LIN {X -214.690,Y 120.896,Z -29.506,A 0.015,B -0.000,C -180.000} C_DIS
LIN {X -218.092,Y 115.236,Z -29.750,A 0.015,B 0.000,C -180.000} C_DIS
LIN {X -214.270,Y 109.850,Z -29.994,A 0.015,B 0.000,C 180.000} C_DIS
LIN {X -207.804,Y 111.194,Z -30.238,A 0.015,B 0.000,C 180.000} C_DIS
LIN {X -206.444,Y 117.657,Z -30.482,A 0.015,B 0.000,C 180.000} C_DIS
LIN {X -211.820,Y 121.492,Z -30.726,A 0.015,B 0.000,C 180.000} C_DIS
LIN {X -217.489,Y 118.103,Z -30.970,A 0.015,B 0.000,C -180.000} C_DIS
LIN {X -216.656,Y 111.552,Z -31.214,A 0.015,B -0.000,C -180.000} C_DIS
LIN {X -210.319,Y 109.690,Z -31.458,A 0.015,B 0.000,C -180.000} C_DIS
LIN {X -206.074,Y 114.749,Z -31.702,A 0.015,B 0.000,C 180.000} C_DIS
LIN {X -209.009,Y 120.666,Z -31.946,A 0.015,B 0.000,C 180.000} C_DIS
LIN {X -215.605,Y 120.349,Z -32.190,A 0.015,B -0.000,C 180.000} C_DIS
LIN {X -217.958,Y 114.177,Z -32.435,A 0.015,B 0.000,C -180.000} C_DIS
LIN {X -213.247,Y 109.549,Z -32.679,A 0.015,B 0.000,C 180.000} C_DIS
LIN {X -207.118,Y 112.011,Z -32.923,A 0.015,B 0.000,C 180.000} C_DIS
LIN {X -206.918,Y 118.612,Z -33.167,A 0.015,B 0.000,C -180.000} C_DIS
LIN {X -212.886,Y 121.441,Z -33.411,A 0.015,B 0.000,C -180.000} C_DIS
LIN {X -217.869,Y 117.107,Z -33.655,A 0.015,B -0.000,C 180.000} C_DIS
LIN {X -215.895,Y 110.804,Z -33.899,A 0.015,B 0.000,C 180.000} C_DIS
LIN {X -209.329,Y 110.088,Z -34.143,A 0.015,B 0.000,C -180.000} C_DIS
LIN {X -206.042,Y 115.816,Z -34.387,A 0.015,B 0.000,C -180.000} C_DIS
LIN {X -209.972,Y 121.123,Z -34.631,A 0.015,B 0.000,C -180.000} C_DIS
LIN {X -216.410,Y 119.648,Z -34.875,A 0.015,B -0.000,C -180.000} C_DIS
LIN {X -217.639,Y 113.160,Z -35.119,A 0.015,B 0.000,C -180.000} C_DIS
LIN {X -212.186,Y 109.433,Z -35.363,A 0.015,B 0.000,C 180.000} C_DIS
LIN {X -206.587,Y 112.936,Z -35.607,A 0.015,B 0.000,C 180.000} C_DIS
LIN {X -207.553,Y 119.469,Z -35.851,A 0.015,B 0.000,C -180.000} C_DIS
LIN {X -213.926,Y 121.203,Z -36.095,A 0.015,B 0.000,C 180.000} C_DIS
LIN {X -218.067,Y 116.059,Z -36.339,A 0.015,B 0.000,C -180.000} C_DIS
LIN {X -215.014,Y 110.203,Z -36.583,A 0.015,B -0.000,C -180.000} C_DIS
LIN {X -208.425,Y 110.653,Z -36.827,A 0.015,B 0.000,C 180.000} C_DIS
LIN {X -206.198,Y 116.871,Z -37.071,A 0.015,B 0.000,C 180.000} C_DIS
LIN {X -211.002,Y 121.403,Z -37.315,A 0.015,B 0.000,C -180.000} C_DIS
LIN {X -217.079,Y 118.818,Z -37.560,A 0.015,B 0.000,C 180.000} C_DIS
LIN {X -217.146,Y 112.214,Z -37.804,A 0.015,B -0.000,C 180.000} C_DIS
LIN {X -211.122,Y 109.506,Z -38.048,A 0.015,B -0.000,C 180.000} C_DIS
LIN {X -206.227,Y 113.940,Z -38.292,A 0.015,B -0.000,C 180.000} C_DIS
LIN {X -208.329,Y 120.201,Z -38.536,A 0.015,B 0.000,C 180.000} C_DIS
LIN {X -214.907,Y 120.785,Z -38.780,A 0.015,B 0.000,C -180.000} C_DIS
LIN {X -218.078,Y 114.992,Z -39.024,A 0.015,B 0.000,C 180.000} C_DIS
LIN {X -214.041,Y 109.765,Z -39.268,A 0.015,B 0.000,C -180.000} C_DIS
LIN {X -207.635,Y 111.369,Z -39.512,A 0.015,B -0.000,C 180.000} C_DIS
LIN {X -206.537,Y 117.882,Z -39.756,A 0.015,B 0.000,C -180.000} C_DIS
LIN {X -212.064,Y 121.497,Z -40.000,A 0.015,B -0.000,C 180.000} C_DIS
LIN {X -214.189,Y 121.497,Z -40.000,A 0.015,B 0.000,C 180.000} C_DIS
CIRC {X -216.111,Y 120.388,Z -40.000,A 0.015,B 0.000,C 180.000},{X -216.113,Y 118.169,Z -40.000,A 0.015,B 0.000,C -180.000} C_DIS
LIN {X -214.876,Y 116.023,Z -40.000,A 0.015,B -0.000,C 180.000} C_DIS
CIRC {X -213.837,Y 114.982,Z -40.000,A 0.015,B 0.000,C -180.000},{X -212.416,Y 114.601,Z -40.000,A 0.015,B -0.000,C 180.000} C_DIS
LIN {X -181.082,Y 114.601,Z -40.000,A 0.015,B 0.000,C -180.000} C_DIS
CIRC {X -179.663,Y 114.981,Z -40.000,A 0.015,B -0.000,C -180.000},{X -178.624,Y 116.020,Z -40.000,A 0.015,B 0.000,C -180.000} C_DIS
LIN {X -177.385,Y 118.164,Z -40.000,A 0.015,B -0.000,C 180.000} C_DIS
CIRC {X -177.385,Y 120.386,Z -40.000,A 0.015,B 0.000,C -180.000},{X -179.309,Y 121.497,Z -40.000,A 0.015,B 0.000,C 180.000} C_DIS
LIN {X -212.064,Y 121.497,Z -40.000,A 0.015,B -0.000,C 180.000} C_DIS
CIRC {X -215.504,Y 122.547,Z -40.000,A 0.015,B 0.000,C -180.000},{X -217.770,Y 125.339,Z -40.000,A 0.015,B 0.000,C 180.000} C_DIS
CIRC {X -219.938,Y 128.171,Z -40.000,A 0.015,B -0.000,C 180.000},{X -223.248,Y 129.500,Z -40.000,A 0.015,B -0.000,C -180.000} C_DIS
CIRC {X -226.517,Y 129.867,Z -40.000,A 0.015,B 0.000,C -180.000},{X -229.788,Y 130.221,Z -40.000,A 0.015,B 0.000,C 180.000} C_DIS
CIRC {X -231.585,Y 129.305,Z -40.000,A 0.015,B -0.000,C 180.000},{X -231.476,Y 127.292,Z -40.000,A 0.015,B -0.000,C -180.000} C_DIS
CIRC {X -228.692,Y 123.319,Z -40.000,A 0.015,B 0.000,C -180.000},{X -226.063,Y 119.242,Z -40.000,A 0.015,B 0.000,C 180.000} C_DIS
CIRC {X -223.545,Y 115.096,Z -40.000,A 0.015,B 0.000,C 180.000},{X -221.091,Y 110.912,Z -40.000,A 0.015,B 0.000,C -180.000} C_DIS
CIRC {X -217.986,Y 107.803,Z -40.000,A 0.015,B 0.000,C 180.000},{X -213.742,Y 106.665,Z -40.000,A 0.015,B 0.000,C 180.000} C_DIS
LIN {X -179.770,Y 106.665,Z -40.000,A 0.015,B 0.000,C -180.000} C_DIS
CIRC {X -175.521,Y 107.803,Z -40.000,A 0.015,B 0.000,C 180.000},{X -172.409,Y 110.912,Z -40.000,A 0.015,B 0.000,C 180.000} C_DIS
CIRC {X -169.958,Y 115.089,Z -40.000,A 0.015,B -0.000,C -180.000},{X -167.450,Y 119.233,Z -40.000,A 0.015,B 0.000,C 180.000} C_DIS
CIRC {X -164.835,Y 123.311,Z -40.000,A 0.015,B 0.000,C -180.000},{X -162.065,Y 127.285,Z -40.000,A 0.015,B 0.000,C -180.000} C_DIS
CIRC {X -161.960,Y 129.301,Z -40.000,A 0.015,B 0.000,C 180.000},{X -163.759,Y 130.217,Z -40.000,A 0.015,B -0.000,C 180.000} C_DIS
CIRC {X -167.466,Y 129.816,Z -40.000,A 0.015,B 0.000,C -180.000},{X -171.172,Y 129.397,Z -40.000,A 0.015,B 0.000,C -180.000} C_DIS
CIRC {X -174.888,Y 129.076,Z -40.000,A 0.015,B 0.000,C 180.000},{X -178.617,Y 128.969,Z -40.000,A 0.015,B 0.000,C -180.000} C_DIS
LIN {X -214.895,Y 128.968,Z -40.000,A 0.015,B 0.000,C -180.000} C_DIS
CIRC {X -218.633,Y 129.075,Z -40.000,A 0.015,B 0.000,C -180.000},{X -222.358,Y 129.398,Z -40.000,A 0.015,B -0.000,C -180.000} C_DIS
LIN {X -223.248,Y 129.500,Z -40.000,A 0.015,B 0.000,C 180.000} C_DIS
CIRC {X -226.419,Y 130.853,Z -40.000,A 0.015,B 0.000,C 180.000},{X -228.335,Y 133.719,Z -40.000,A 0.015,B -0.000,C 180.000} C_DIS
CIRC {X -230.253,Y 136.582,Z -40.000,A 0.015,B 0.000,C -180.000},{X -233.421,Y 137.938,Z -40.000,A 0.015,B 0.000,C -180.000} C_DIS
CIRC {X -237.034,Y 138.381,Z -40.000,A 0.015,B 0.000,C 180.000},{X -240.642,Y 138.863,Z -40.000,A 0.015,B 0.000,C 180.000} C_DIS
CIRC {X -242.321,Y 139.135,Z -40.000,A 0.015,B 0.000,C -180.000},{X -243.987,Y 139.480,Z -40.000,A 0.015,B 0.000,C 180.000} C_DIS
CIRC {X -245.648,Y 139.845,Z -40.000,A 0.015,B -0.000,C -180.000},{X -247.316,Y 140.180,Z -40.000,A 0.015,B 0.000,C 180.000} C_DIS
CIRC {X -249.035,Y 139.393,Z -40.000,A 0.015,B 0.000,C -180.000},{X -248.855,Y 137.511,Z -40.000,A 0.015,B -0.000,C -180.000} C_DIS
LIN {X -243.268,Y 131.116,Z -40.000,A 0.015,B 0.000,C -180.000} C_DIS
CIRC {X -240.525,Y 127.874,Z -40.000,A 0.015,B -0.000,C 180.000},{X -237.914,Y 124.524,Z -40.000,A 0.015,B 0.000,C -180.000} C_DIS
CIRC {X -234.428,Y 119.496,Z -40.000,A 0.015,B -0.000,C -180.000},{X -231.314,Y 114.230,Z -40.000,A 0.015,B -0.000,C -180.000} C_DIS
CIRC {X -228.360,Y 108.876,Z -40.000,A 0.015,B 0.000,C -180.000},{X -225.339,Y 103.559,Z -40.000,A 0.015,B -0.000,C -180.000} C_DIS
CIRC {X -222.234,Y 100.451,Z -40.000,A 0.015,B -0.000,C -180.000},{X -217.991,Y 99.313,Z -40.000,A 0.015,B 0.000,C -180.000} C_DIS
LIN {X -175.527,Y 99.313,Z -40.000,A 0.015,B 0.000,C 180.000} C_DIS
CIRC {X -171.278,Y 100.451,Z -40.000,A 0.015,B 0.000,C 180.000},{X -168.166,Y 103.560,Z -40.000,A 0.015,B 0.000,C -180.000} C_DIS
CIRC {X -167.080,Y 105.510,Z -40.000,A 0.015,B 0.000,C -180.000},{X -166.055,Y 107.493,Z -40.000,A 0.015,B 0.000,C 180.000} C_DIS
CIRC {X -165.030,Y 109.476,Z -40.000,A 0.015,B -0.000,C 180.000},{X -163.943,Y 111.426,Z -40.000,A 0.015,B 0.000,C 180.000} C_DIS
CIRC {X -159.653,Y 118.326,Z -40.000,A 0.015,B 0.000,C 180.000},{X -154.928,Y 124.936,Z -40.000,A 0.015,B -0.000,C 180.000} C_DIS
CIRC {X -149.891,Y 131.308,Z -40.000,A 0.015,B -0.000,C 180.000},{X -144.653,Y 137.515,Z -40.000,A 0.015,B 0.000,C 180.000} C_DIS
CIRC {X -144.469,Y 139.395,Z -40.000,A 0.015,B 0.000,C -180.000},{X -146.185,Y 140.182,Z -40.000,A 0.015,B 0.000,C 180.000} C_DIS
CIRC {X -169.667,Y 136.815,Z -40.000,A 0.015,B 0.000,C -180.000},{X -193.359,Y 135.650,Z -40.000,A 0.015,B -0.000,C 180.000} C_DIS
CIRC {X -213.424,Y 136.197,Z -40.000,A 0.015,B -0.000,C 180.000},{X -233.421,Y 137.938,Z -40.000,A 0.015,B 0.000,C -180.000} C_DIS
CIRC {X -236.184,Y 139.158,Z -40.000,A 0.015,B 0.000,C 180.000},{X -237.779,Y 141.722,Z -40.000,A 0.015,B -0.000,C -180.000} C_DIS
CIRC {X -239.318,Y 144.301,Z -40.000,A 0.015,B 0.000,C -180.000},{X -241.992,Y 145.667,Z -40.000,A 0.015,B 0.000,C -180.000} C_DIS
CIRC {X -243.728,Y 146.016,Z -40.000,A 0.015,B 0.000,C 180.000},{X -245.460,Y 146.386,Z -40.000,A 0.015,B 0.000,C 180.000} C_DIS
CIRC {X -260.324,Y 150.371,Z -40.000,A 0.015,B -0.000,C 180.000},{X -274.770,Y 155.672,Z -40.000,A 0.015,B 0.000,C 180.000} C_DIS
CIRC {X -276.326,Y 155.146,Z -40.000,A 0.015,B 0.000,C -180.000},{X -275.997,Y 153.536,Z -40.000,A 0.015,B 0.000,C -180.000} C_DIS
CIRC {X -266.962,Y 146.173,Z -40.000,A 0.015,B 0.000,C -180.000},{X -258.508,Y 138.148,Z -40.000,A 0.015,B 0.000,C -180.000} C_DIS
CIRC {X -250.643,Y 129.549,Z -40.000,A 0.015,B 0.000,C 180.000},{X -243.360,Y 120.451,Z -40.000,A 0.015,B 0.000,C 180.000} C_DIS
CIRC {X -241.141,Y 117.355,Z -40.000,A 0.015,B 0.000,C -180.000},{X -239.047,Y 114.173,Z -40.000,A 0.015,B 0.000,C -180.000} C_DIS
CIRC {X -237.049,Y 110.931,Z -40.000,A 0.015,B 0.000,C -180.000},{X -235.115,Y 107.650,Z -40.000,A 0.015,B -0.000,C 180.000} C_DIS
CIRC {X -233.613,Y 104.946,Z -40.000,A 0.015,B -0.000,C 180.000},{X -232.196,Y 102.197,Z -40.000,A 0.015,B -0.000,C -180.000} C_DIS
CIRC {X -230.779,Y 99.448,Z -40.000,A 0.015,B 0.000,C -180.000},{X -229.277,Y 96.745,Z -40.000,A 0.015,B -0.000,C -180.000} C_DIS
CIRC {X -226.172,Y 93.636,Z -40.000,A 0.015,B -0.000,C -180.000},{X -221.929,Y 92.498,Z -40.000,A 0.015,B 0.000,C 180.000} C_DIS
LIN {X -171.595,Y 92.498,Z -40.000,A 0.015,B -0.000,C 180.000} C_DIS
CIRC {X -167.346,Y 93.636,Z -40.000,A 0.015,B 0.000,C 180.000},{X -164.234,Y 96.746,Z -40.000,A 0.015,B 0.000,C -180.000} C_DIS
CIRC {X -162.669,Y 99.555,Z -40.000,A 0.015,B -0.000,C 180.000},{X -161.192,Y 102.412,Z -40.000,A 0.015,B -0.000,C -180.000} C_DIS
CIRC {X -159.715,Y 105.268,Z -40.000,A 0.015,B 0.000,C 180.000},{X -158.150,Y 108.078,Z -40.000,A 0.015,B 0.000,C 180.000} C_DIS
CIRC {X -149.768,Y 120.946,Z -40.000,A 0.015,B 0.000,C -180.000},{X -140.064,Y 132.849,Z -40.000,A 0.015,B -0.000,C 180.000} C_DIS
CIRC {X -129.235,Y 143.731,Z -40.000,A 0.015,B 0.000,C 180.000},{X -117.456,Y 153.577,Z -40.000,A 0.015,B 0.000,C 180.000} C_DIS
CIRC {X -117.135,Y 155.187,Z -40.000,A 0.015,B 0.000,C -180.000},{X -118.693,Y 155.704,Z -40.000,A 0.015,B 0.000,C -180.000} C_DIS
CIRC {X -128.956,Y 151.768,Z -40.000,A 0.015,B -0.000,C 180.000},{X -139.478,Y 148.589,Z -40.000,A 0.015,B 0.000,C 180.000} C_DIS
CIRC {X -150.185,Y 146.112,Z -40.000,A 0.015,B 0.000,C 180.000},{X -161.020,Y 144.276,Z -40.000,A 0.015,B 0.000,C 180.000} C_DIS
CIRC {X -169.797,Y 143.362,Z -40.000,A 0.015,B -0.000,C -180.000},{X -178.617,Y 143.057,Z -40.000,A 0.015,B -0.000,C -180.000} C_DIS
LIN {X -214.895,Y 143.057,Z -40.000,A 0.015,B 0.000,C 180.000} C_DIS
CIRC {X -228.506,Y 143.711,Z -40.000,A 0.015,B 0.000,C 180.000},{X -241.992,Y 145.667,Z -40.000,A 0.015,B 0.000,C -180.000} C_DIS
CIRC {X -244.741,Y 147.123,Z -40.000,A 0.015,B 0.000,C 180.000},{X -246.215,Y 149.862,Z -40.000,A 0.015,B 0.000,C -180.000} C_DIS
CIRC {X -247.650,Y 152.609,Z -40.000,A 0.015,B 0.000,C 180.000},{X -250.334,Y 154.160,Z -40.000,A 0.015,B 0.000,C 180.000} C_DIS
CIRC {X -257.545,Y 156.101,Z -40.000,A 0.015,B -0.000,C 180.000},{X -264.665,Y 158.353,Z -40.000,A 0.015,B 0.000,C -180.000} C_DIS
CIRC {X -269.256,Y 160.100,Z -40.000,A 0.015,B 0.000,C 180.000},{X -273.710,Y 162.168,Z -40.000,A 0.015,B -0.000,C -180.000} C_DIS
LIN {X -283.276,Y 167.029,Z -40.000,A 0.015,B -0.000,C -180.000} C_DIS
CIRC {X -285.545,Y 166.939,Z -40.000,A 0.015,B 0.000,C 180.000},{X -286.654,Y 164.957,Z -40.000,A 0.015,B 0.000,C -180.000} C_DIS
LIN {X -286.654,Y 156.539,Z -40.000,A 0.015,B 0.000,C -180.000} C_DIS
CIRC {X -285.883,Y 153.392,Z -40.000,A 0.015,B 0.000,C 180.000},{X -283.747,Y 150.958,Z -40.000,A 0.015,B 0.000,C 180.000} C_DIS
CIRC {X -271.170,Y 141.133,Z -40.000,A 0.015,B 0.000,C -180.000},{X -259.697,Y 130.038,Z -40.000,A 0.015,B 0.000,C -180.000} C_DIS
CIRC {X -249.502,Y 117.754,Z -40.000,A 0.015,B 0.000,C -180.000},{X -240.761,Y 104.396,Z -40.000,A 0.015,B 0.000,C 180.000} C_DIS
CIRC {X -238.793,Y 100.854,Z -40.000,A 0.015,B 0.000,C 180.000},{X -236.936,Y 97.253,Z -40.000,A 0.015,B 0.000,C 180.000} C_DIS
CIRC {X -235.080,Y 93.651,Z -40.000,A 0.015,B -0.000,C -180.000},{X -233.112,Y 90.109,Z -40.000,A 0.015,B 0.000,C -180.000} C_DIS
CIRC {X -230.007,Y 87.001,Z -40.000,A 0.015,B 0.000,C 180.000},{X -225.763,Y 85.863,Z -40.000,A 0.015,B 0.000,C 180.000} C_DIS
LIN {X -167.766,Y 85.863,Z -40.000,A 0.015,B 0.000,C 180.000} C_DIS
CIRC {X -163.516,Y 87.001,Z -40.000,A 0.015,B 0.000,C 180.000},{X -160.405,Y 90.110,Z -40.000,A 0.015,B 0.000,C 180.000} C_DIS
CIRC {X -158.373,Y 93.756,Z -40.000,A 0.015,B 0.000,C 180.000},{X -156.456,Y 97.464,Z -40.000,A 0.015,B 0.000,C -180.000} C_DIS
CIRC {X -154.540,Y 101.171,Z -40.000,A 0.015,B 0.000,C -180.000},{X -152.508,Y 104.817,Z -40.000,A 0.015,B 0.000,C 180.000} C_DIS
CIRC {X -143.805,Y 118.066,Z -40.000,A 0.015,B 0.000,C -180.000},{X -133.646,Y 130.234,Z -40.000,A 0.015,B -0.000,C 180.000} C_DIS
CIRC {X -122.233,Y 141.226,Z -40.000,A 0.015,B 0.000,C -180.000},{X -109.753,Y 150.992,Z -40.000,A 0.015,B 0.000,C 180.000} C_DIS
CIRC {X -107.625,Y 153.424,Z -40.000,A 0.015,B 0.000,C 180.000},{X -106.858,Y 156.564,Z -40.000,A 0.015,B -0.000,C 180.000} C_DIS
LIN {X -106.859,Y 164.937,Z -40.000,A 0.015,B 0.000,C -180.000} C_DIS
CIRC {X -107.968,Y 166.911,Z -40.000,A 0.015,B 0.000,C 180.000},{X -110.230,Y 166.990,Z -40.000,A 0.015,B -0.000,C 180.000} C_DIS
CIRC {X -122.583,Y 161.292,Z -40.000,A 0.015,B 0.000,C 180.000},{X -135.397,Y 156.724,Z -40.000,A 0.015,B -0.000,C -180.000} C_DIS
CIRC {X -148.548,Y 153.257,Z -40.000,A 0.015,B 0.000,C -180.000},{X -161.934,Y 150.848,Z -40.000,A 0.015,B 0.000,C 180.000} C_DIS
CIRC {X -170.255,Y 149.982,Z -40.000,A 0.015,B 0.000,C 180.000},{X -178.617,Y 149.693,Z -40.000,A 0.015,B 0.000,C -180.000} C_DIS
LIN {X -214.895,Y 149.693,Z -40.000,A 0.015,B 0.000,C 180.000} C_DIS
CIRC {X -227.567,Y 150.265,Z -40.000,A 0.015,B -0.000,C -180.000},{X -240.136,Y 151.977,Z -40.000,A 0.015,B 0.000,C -180.000} C_DIS
CIRC {X -245.252,Y 152.991,Z -40.000,A 0.015,B 0.000,C 180.000},{X -250.334,Y 154.160,Z -40.000,A 0.015,B -0.000,C 180.000} C_DIS
CIRC {X -253.660,Y 156.157,Z -40.000,A 0.015,B -0.000,C 180.000},{X -255.280,Y 159.681,Z -40.000,A 0.015,B -0.000,C -180.000} C_DIS
CIRC {X -256.805,Y 163.218,Z -40.000,A 0.015,B 0.000,C 180.000},{X -259.959,Y 165.430,Z -40.000,A 0.015,B -0.000,C 180.000} C_DIS
CIRC {X -276.245,Y 172.320,Z -40.000,A 0.015,B 0.000,C 180.000},{X -291.506,Y 181.253,Z -40.000,A 0.015,B 0.000,C -180.000} C_DIS
CIRC {X -293.652,Y 181.365,Z -40.000,A 0.015,B -0.000,C -180.000},{X -294.758,Y 179.523,Z -40.000,A 0.015,B 0.000,C 180.000} C_DIS
LIN {X -294.757,Y 153.804,Z -40.000,A 0.015,B 0.000,C 180.000} C_DIS
CIRC {X -293.661,Y 149.334,Z -40.000,A 0.015,B -0.000,C -180.000},{X -290.622,Y 145.877,Z -40.000,A 0.015,B 0.000,C 180.000} C_DIS
CIRC {X -286.379,Y 142.894,Z -40.000,A 0.015,B 0.000,C 180.000},{X -282.158,Y 139.879,Z -40.000,A 0.015,B 0.000,C 180.000} C_DIS
CIRC {X -278.036,Y 136.728,Z -40.000,A 0.015,B 0.000,C -180.000},{X -274.099,Y 133.347,Z -40.000,A 0.015,B -0.000,C 180.000} C_DIS
CIRC {X -268.929,Y 128.312,Z -40.000,A 0.015,B -0.000,C -180.000},{X -264.114,Y 122.936,Z -40.000,A 0.015,B 0.000,C 180.000} C_DIS
CIRC {X -259.562,Y 117.340,Z -40.000,A 0.015,B 0.000,C 180.000},{X -255.164,Y 111.623,Z -40.000,A 0.015,B 0.000,C -180.000} C_DIS
CIRC {X -251.289,Y 106.107,Z -40.000,A 0.015,B 0.000,C 180.000},{X -247.750,Y 100.369,Z -40.000,A 0.015,B 0.000,C -180.000} C_DIS
CIRC {X -245.202,Y 95.810,Z -40.000,A 0.015,B -0.000,C 180.000},{X -242.773,Y 91.187,Z -40.000,A 0.015,B 0.000,C 180.000} C_DIS
CIRC {X -240.344,Y 86.564,Z -40.000,A 0.015,B 0.000,C -180.000},{X -237.795,Y 82.006,Z -40.000,A 0.015,B -0.000,C -180.000} C_DIS
CIRC {X -234.690,Y 78.897,Z -40.000,A 0.015,B 0.000,C -180.000},{X -230.446,Y 77.759,Z -40.000,A 0.015,B 0.000,C 180.000} C_DIS
LIN {X -163.089,Y 77.759,Z -40.000,A 0.015,B 0.000,C 180.000} C_DIS
CIRC {X -158.840,Y 78.897,Z -40.000,A 0.015,B 0.000,C -180.000},{X -155.728,Y 82.007,Z -40.000,A 0.015,B 0.000,C -180.000} C_DIS
CIRC {X -153.114,Y 86.666,Z -40.000,A 0.015,B 0.000,C -180.000},{X -150.619,Y 91.390,Z -40.000,A 0.015,B -0.000,C 180.000} C_DIS
CIRC {X -148.124,Y 96.114,Z -40.000,A 0.015,B -0.000,C 180.000},{X -145.510,Y 100.773,Z -40.000,A 0.015,B 0.000,C 180.000} C_DIS
CIRC {X -136.917,Y 113.796,Z -40.000,A 0.015,B 0.000,C -180.000},{X -126.846,Y 125.713,Z -40.000,A 0.015,B 0.000,C 180.000} C_DIS
CIRC {X -115.486,Y 136.403,Z -40.000,A 0.015,B 0.000,C -180.000},{X -103.022,Y 145.783,Z -40.000,A 0.015,B 0.000,C 180.000} C_DIS
CIRC {X -99.888,Y 149.247,Z -40.000,A 0.015,B 0.000,C -180.000},{X -98.755,Y 153.779,Z -40.000,A 0.015,B 0.000,C -180.000} C_DIS
LIN {X -98.755,Y 179.510,Z -40.000,A 0.015,B 0.000,C 180.000} C_DIS
CIRC {X -99.862,Y 181.369,Z -40.000,A 0.015,B 0.000,C 180.000},{X -102.023,Y 181.282,Z -40.000,A 0.015,B 0.000,C -180.000} C_DIS
CIRC {X -110.211,Y 176.258,Z -40.000,A 0.015,B 0.000,C 180.000},{X -118.658,Y 171.685,Z -40.000,A 0.015,B -0.000,C 180.000} C_DIS
CIRC {X -127.391,Y 167.675,Z -40.000,A 0.015,B 0.000,C 180.000},{X -136.407,Y 164.351,Z -40.000,A 0.015,B 0.000,C -180.000} C_DIS
CIRC {X -155.656,Y 159.675,Z -40.000,A 0.015,B 0.000,C -180.000},{X -175.393,Y 157.980,Z -40.000,A 0.015,B 0.000,C -180.000} C_DIS
LIN {X -214.895,Y 157.797,Z -40.000,A 0.015,B -0.000,C 180.000} C_DIS
CIRC {X -237.748,Y 159.718,Z -40.000,A 0.015,B -0.000,C 180.000},{X -259.959,Y 165.430,Z -40.000,A 0.015,B 0.000,C 180.000} C_DIS
CIRC {X -262.962,Y 167.626,Z -40.000,A 0.015,B -0.000,C 180.000},{X -264.228,Y 171.125,Z -40.000,A 0.015,B 0.000,C -180.000} C_DIS
CIRC {X -265.425,Y 174.627,Z -40.000,A 0.015,B 0.000,C 180.000},{X -268.291,Y 176.970,Z -40.000,A 0.015,B 0.000,C 180.000} C_DIS
CIRC {X -272.041,Y 178.652,Z -40.000,A 0.015,B 0.000,C 180.000},{X -275.743,Y 180.440,Z -40.000,A 0.015,B 0.000,C 180.000} C_DIS
CIRC {X -282.030,Y 183.929,Z -40.000,A 0.015,B 0.000,C 180.000},{X -287.996,Y 187.941,Z -40.000,A 0.015,B 0.000,C -180.000} C_DIS
CIRC {X -293.740,Y 192.257,Z -40.000,A 0.015,B 0.000,C 180.000},{X -299.397,Y 196.684,Z -40.000,A 0.015,B 0.000,C 180.000} C_DIS
CIRC {X -301.459,Y 196.918,Z -40.000,A 0.015,B 0.000,C 180.000},{X -302.564,Y 195.161,Z -40.000,A 0.015,B -0.000,C -180.000} C_DIS
LIN {X -302.562,Y 149.253,Z -40.000,A 0.015,B 0.000,C -180.000} C_DIS
CIRC {X -301.466,Y 144.963,Z -40.000,A 0.015,B 0.000,C -180.000},{X -298.447,Y 141.724,Z -40.000,A 0.015,B 0.000,C 180.000} C_DIS
CIRC {X -288.038,Y 134.334,Z -40.000,A 0.015,B -0.000,C 180.000},{X -278.369,Y 125.999,Z -40.000,A 0.015,B 0.000,C 180.000} C_DIS
CIRC {X -269.486,Y 116.835,Z -40.000,A 0.015,B -0.000,C 180.000},{X -261.414,Y 106.948,Z -40.000,A 0.015,B 0.000,C 180.000} C_DIS
CIRC {X -257.807,Y 101.813,Z -40.000,A 0.015,B 0.000,C 180.000},{X -254.513,Y 96.472,Z -40.000,A 0.015,B 0.000,C 180.000} C_DIS
CIRC {X -251.402,Y 90.936,Z -40.000,A 0.015,B -0.000,C -180.000},{X -248.409,Y 85.336,Z -40.000,A 0.015,B -0.000,C 180.000} C_DIS
CIRC {X -245.417,Y 79.736,Z -40.000,A 0.015,B -0.000,C 180.000},{X -242.306,Y 74.201,Z -40.000,A 0.015,B 0.000,C 180.000} C_DIS
CIRC {X -239.201,Y 71.092,Z -40.000,A 0.015,B 0.000,C -180.000},{X -234.957,Y 69.954,Z -40.000,A 0.015,B 0.000,C 180.000} C_DIS
LIN {X -158.585,Y 69.954,Z -40.000,A 0.015,B 0.000,C 180.000} C_DIS
CIRC {X -154.336,Y 71.092,Z -40.000,A 0.015,B 0.000,C 180.000},{X -151.224,Y 74.201,Z -40.000,A 0.015,B -0.000,C 180.000} C_DIS
LIN {X -138.752,Y 96.868,Z -40.000,A 0.015,B -0.000,C -180.000} C_DIS
CIRC {X -130.141,Y 109.762,Z -40.000,A 0.015,B 0.000,C -180.000},{X -119.937,Y 121.436,Z -40.000,A 0.015,B 0.000,C 180.000} C_DIS
CIRC {X -108.478,Y 131.862,Z -40.000,A 0.015,B 0.000,C 180.000},{X -96.045,Y 141.103,Z -40.000,A 0.015,B 0.000,C -180.000} C_DIS
LIN {X -95.557,Y 141.407,Z -40.000,A 0.015,B -0.000,C 180.000} C_DIS
LIN {X -95.066,Y 141.708,Z -40.000,A 0.015,B 0.000,C 180.000} C_DIS
CIRC {X -92.045,Y 144.990,Z -40.000,A 0.015,B 0.000,C 180.000},{X -90.949,Y 149.315,Z -40.000,A 0.015,B 0.000,C 180.000} C_DIS
LIN {X -90.951,Y 195.181,Z -40.000,A 0.015,B 0.000,C 180.000} C_DIS
CIRC {X -92.055,Y 196.943,Z -40.000,A 0.015,B -0.000,C 180.000},{X -94.122,Y 196.716,Z -40.000,A 0.015,B 0.000,C 180.000} C_DIS
CIRC {X -101.310,Y 191.252,Z -40.000,A 0.015,B 0.000,C -180.000},{X -108.704,Y 186.071,Z -40.000,A 0.015,B -0.000,C 180.000} C_DIS
CIRC {X -116.396,Y 181.333,Z -40.000,A 0.015,B -0.000,C 180.000},{X -124.441,Y 177.222,Z -40.000,A 0.015,B 0.000,C 180.000} C_DIS
CIRC {X -134.001,Y 173.361,Z -40.000,A 0.015,B -0.000,C 180.000},{X -143.892,Y 170.451,Z -40.000,A 0.015,B 0.000,C 180.000} C_DIS
CIRC {X -153.962,Y 168.277,Z -40.000,A 0.015,B 0.000,C 180.000},{X -164.126,Y 166.605,Z -40.000,A 0.015,B 0.000,C 180.000} C_DIS
CIRC {X -171.354,Y 165.853,Z -40.000,A 0.015,B 0.000,C -180.000},{X -178.617,Y 165.602,Z -40.000,A 0.015,B 0.000,C -180.000} C_DIS
LIN {X -214.895,Y 165.602,Z -40.000,A 0.015,B 0.000,C 180.000} C_DIS
CIRC {X -230.659,Y 166.574,Z -40.000,A 0.015,B 0.000,C 180.000},{X -246.184,Y 169.475,Z -40.000,A 0.015,B -0.000,C -180.000} C_DIS
CIRC {X -257.388,Y 172.777,Z -40.000,A 0.015,B 0.000,C 180.000},{X -268.291,Y 176.970,Z -40.000,A 0.015,B 0.000,C 180.000} C_DIS
CIRC {X -271.061,Y 179.343,Z -40.000,A 0.015,B -0.000,C -180.000},{X -272.000,Y 182.868,Z -40.000,A 0.015,B 0.000,C -180.000} C_DIS
CIRC {X -272.841,Y 186.389,Z -40.000,A 0.015,B 0.000,C 180.000},{X -275.400,Y 188.950,Z -40.000,A 0.015,B 0.000,C -180.000} C_DIS
CIRC {X -292.319,Y 200.359,Z -40.000,A 0.015,B -0.000,C -180.000},{X -307.135,Y 214.394,Z -40.000,A 0.015,B 0.000,C 180.000} C_DIS
CIRC {X -309.015,Y 214.857,Z -40.000,A 0.015,B 0.000,C 180.000},{X -310.116,Y 213.263,Z -40.000,A 0.015,B -0.000,C -180.000} C_DIS
LIN {X -310.114,Y 144.714,Z -40.000,A 0.015,B 0.000,C -180.000} C_DIS
CIRC {X -309.001,Y 140.539,Z -40.000,A 0.015,B -0.000,C 180.000},{X -305.958,Y 137.471,Z -40.000,A 0.015,B -0.000,C -180.000} C_DIS
CIRC {X -295.027,Y 130.251,Z -40.000,A 0.015,B 0.000,C 180.000},{X -284.953,Y 121.878,Z -40.000,A 0.015,B -0.000,C 180.000} C_DIS
CIRC {X -275.768,Y 112.547,Z -40.000,A 0.015,B 0.000,C 180.000},{X -267.461,Y 102.426,Z -40.000,A 0.015,B 0.000,C 180.000} C_DIS
CIRC {X -264.114,Y 97.659,Z -40.000,A 0.015,B 0.000,C -180.000},{X -261.056,Y 92.701,Z -40.000,A 0.015,B -0.000,C 180.000} C_DIS
LIN {X -246.670,Y 66.649,Z -40.000,A 0.015,B 0.000,C -180.000} C_DIS
CIRC {X -243.565,Y 63.540,Z -40.000,A 0.015,B 0.000,C -180.000},{X -239.321,Y 62.402,Z -40.000,A 0.015,B 0.000,C 180.000} C_DIS
LIN {X -154.227,Y 62.402,Z -40.000,A 0.015,B -0.000,C 180.000} C_DIS
CIRC {X -149.978,Y 63.540,Z -40.000,A 0.015,B 0.000,C 180.000},{X -146.866,Y 66.650,Z -40.000,A 0.015,B 0.000,C 180.000} C_DIS
LIN {X -132.214,Y 93.089,Z -40.000,A 0.015,B 0.000,C -180.000} C_DIS
CIRC {X -123.318,Y 106.303,Z -40.000,A 0.015,B 0.000,C 180.000},{X -112.701,Y 118.178,Z -40.000,A 0.015,B 0.000,C 180.000} C_DIS
CIRC {X -100.668,Y 128.600,Z -40.000,A 0.015,B 0.000,C -180.000},{X -87.492,Y 137.534,Z -40.000,A 0.015,B -0.000,C -180.000} C_DIS
CIRC {X -84.493,Y 140.594,Z -40.000,A 0.015,B 0.000,C -180.000},{X -83.398,Y 144.736,Z -40.000,A 0.015,B 0.000,C -180.000} C_DIS
LIN {X -83.400,Y 213.259,Z -40.000,A 0.015,B 0.000,C -180.000} C_DIS
CIRC {X -84.500,Y 214.853,Z -40.000,A 0.015,B 0.000,C 180.000},{X -86.381,Y 214.390,Z -40.000,A 0.015,B -0.000,C 180.000} C_DIS
CIRC {X -98.149,Y 202.832,Z -40.000,A 0.015,B 0.000,C 180.000},{X -111.404,Y 193.014,Z -40.000,A 0.015,B 0.000,C -180.000} C_DIS
CIRC {X -125.835,Y 185.039,Z -40.000,A 0.015,B 0.000,C -180.000},{X -141.159,Y 178.954,Z -40.000,A 0.015,B 0.000,C -180.000} C_DIS
CIRC {X -159.214,Y 174.612,Z -40.000,A 0.015,B 0.000,C 180.000},{X -177.725,Y 173.153,Z -40.000,A 0.015,B 0.000,C 180.000} C_DIS
LIN {X -214.895,Y 173.153,Z -40.000,A 0.015,B 0.000,C 180.000} C_DIS
CIRC {X -246.162,Y 177.168,Z -40.000,A 0.015,B 0.000,C 180.000},{X -275.400,Y 188.950,Z -40.000,A 0.015,B -0.000,C 180.000} C_DIS
CIRC {X -277.772,Y 191.437,Z -40.000,A 0.015,B 0.000,C -180.000},{X -278.335,Y 194.828,Z -40.000,A 0.015,B 0.000,C 180.000} C_DIS
CIRC {X -278.819,Y 198.208,Z -40.000,A 0.015,B 0.000,C 180.000},{X -281.003,Y 200.832,Z -40.000,A 0.015,B 0.000,C 180.000} C_DIS
CIRC {X -299.481,Y 216.465,Z -40.000,A 0.015,B 0.000,C 180.000},{X -314.434,Y 235.497,Z -40.000,A 0.015,B 0.000,C 180.000} C_DIS
CIRC {X -316.141,Y 236.143,Z -40.000,A 0.015,B 0.000,C -180.000},{X -317.237,Y 234.683,Z -40.000,A 0.015,B 0.000,C -180.000} C_DIS
LIN {X -317.235,Y 140.248,Z -40.000,A 0.015,B 0.000,C -180.000} C_DIS
CIRC {X -316.140,Y 136.253,Z -40.000,A 0.015,B 0.000,C 180.000},{X -313.163,Y 133.373,Z -40.000,A 0.015,B -0.000,C -180.000} C_DIS
CIRC {X -302.924,Y 127.100,Z -40.000,A 0.015,B 0.000,C 180.000},{X -293.337,Y 119.870,Z -40.000,A 0.015,B 0.000,C 180.000} C_DIS
CIRC {X -284.520,Y 111.716,Z -40.000,A 0.015,B 0.000,C -180.000},{X -276.595,Y 102.693,Z -40.000,A 0.015,B 0.000,C 180.000} C_DIS
CIRC {X -269.249,Y 92.450,Z -40.000,A 0.015,B 0.000,C 180.000},{X -262.891,Y 81.566,Z -40.000,A 0.015,B 0.000,C -180.000} C_DIS
CIRC {X -256.941,Y 70.468,Z -40.000,A 0.015,B 0.000,C -180.000},{X -250.766,Y 59.494,Z -40.000,A 0.015,B 0.000,C -180.000} C_DIS
CIRC {X -247.686,Y 56.410,Z -40.000,A 0.015,B 0.000,C -180.000},{X -243.475,Y 55.281,Z -40.000,A 0.015,B 0.000,C -180.000} C_DIS
LIN {X -150.053,Y 55.281,Z -40.000,A 0.015,B 0.000,C 180.000} C_DIS
CIRC {X -145.860,Y 56.404,Z -40.000,A 0.015,B 0.000,C -180.000},{X -142.789,Y 59.473,Z -40.000,A 0.015,B -0.000,C 180.000} C_DIS
LIN {X -126.048,Y 89.526,Z -40.000,A 0.015,B 0.000,C -180.000} C_DIS
CIRC {X -117.054,Y 102.798,Z -40.000,A 0.015,B 0.000,C 180.000},{X -106.258,Y 114.650,Z -40.000,A 0.015,B -0.000,C -180.000} C_DIS
CIRC {X -93.931,Y 124.893,Z -40.000,A 0.015,B 0.000,C 180.000},{X -80.345,Y 133.396,Z -40.000,A 0.015,B 0.000,C -180.000} C_DIS
CIRC {X -77.371,Y 136.233,Z -40.000,A 0.015,B -0.000,C 180.000},{X -76.276,Y 140.194,Z -40.000,A 0.015,B 0.000,C -180.000} C_DIS
LIN {X -76.279,Y 234.676,Z -40.000,A 0.015,B 0.000,C 180.000} C_DIS
CIRC {X -77.375,Y 236.136,Z -40.000,A 0.015,B 0.000,C -180.000},{X -79.083,Y 235.489,Z -40.000,A 0.015,B 0.000,C -180.000} C_DIS
CIRC {X -106.859,Y 204.970,Z -40.000,A 0.015,B 0.000,C 180.000},{X -143.363,Y 185.725,Z -40.000,A 0.015,B 0.000,C -180.000} C_DIS
CIRC {X -160.917,Y 181.529,Z -40.000,A 0.015,B 0.000,C -180.000},{X -178.914,Y 180.181,Z -40.000,A 0.015,B 0.000,C 180.000} C_DIS
LIN {X -214.895,Y 180.275,Z -40.000,A 0.015,B 0.000,C 180.000} C_DIS
CIRC {X -244.278,Y 184.041,Z -40.000,A 0.015,B 0.000,C -180.000},{X -271.760,Y 195.096,Z -40.000,A 0.015,B 0.000,C -180.000} C_DIS
CIRC {X -276.447,Y 197.859,Z -40.000,A 0.015,B -0.000,C -180.000},{X -281.003,Y 200.832,Z -40.000,A 0.015,B 0.000,C 180.000} C_DIS
CIRC {X -282.988,Y 203.320,Z -40.000,A 0.015,B -0.000,C 180.000},{X -283.243,Y 206.492,Z -40.000,A 0.015,B 0.000,C -180.000} C_DIS
CIRC {X -283.437,Y 209.650,Z -40.000,A 0.015,B 0.000,C 180.000},{X -285.265,Y 212.233,Z -40.000,A 0.015,B 0.000,C 180.000} C_DIS
CIRC {X -293.647,Y 219.640,Z -40.000,A 0.015,B 0.000,C -180.000},{X -301.303,Y 227.795,Z -40.000,A 0.015,B 0.000,C -180.000} C_DIS
CIRC {X -306.526,Y 234.564,Z -40.000,A 0.015,B 0.000,C 180.000},{X -311.046,Y 241.823,Z -40.000,A 0.015,B -0.000,C -180.000} C_DIS
CIRC {X -314.945,Y 249.425,Z -40.000,A 0.015,B 0.000,C -180.000},{X -318.336,Y 257.267,Z -40.000,A 0.015,B -0.000,C 180.000} C_DIS
CIRC {X -321.507,Y 259.015,Z -40.000,A 0.015,B 0.000,C 180.000},{X -323.816,Y 256.227,Z -40.000,A 0.015,B 0.000,C -180.000} C_DIS
LIN {X -323.812,Y 135.870,Z -40.000,A 0.015,B -0.000,C 180.000} C_DIS
CIRC {X -322.718,Y 132.050,Z -40.000,A 0.015,B -0.000,C -180.000},{X -319.767,Y 129.389,Z -40.000,A 0.015,B 0.000,C -180.000} C_DIS
CIRC {X -299.017,Y 116.156,Z -40.000,A 0.015,B 0.000,C -180.000},{X -281.755,Y 98.615,Z -40.000,A 0.015,B 0.000,C 180.000} C_DIS
CIRC {X -273.958,Y 87.766,Z -40.000,A 0.015,B -0.000,C 180.000},{X -267.182,Y 76.251,Z -40.000,A 0.015,B -0.000,C -180.000} C_DIS
LIN {X -254.496,Y 52.765,Z -40.000,A 0.015,B -0.000,C 180.000} C_DIS
CIRC {X -251.611,Y 49.794,Z -40.000,A 0.015,B 0.000,C 180.000},{X -247.616,Y 48.703,Z -40.000,A 0.015,B 0.000,C -180.000} C_DIS
LIN {X -145.879,Y 48.703,Z -40.000,A 0.015,B -0.000,C 180.000} C_DIS
CIRC {X -141.902,Y 49.795,Z -40.000,A 0.015,B 0.000,C 180.000},{X -139.040,Y 52.763,Z -40.000,A 0.015,B 0.000,C -180.000} C_DIS
LIN {X -119.938,Y 86.414,Z -40.000,A 0.015,B 0.000,C 180.000} C_DIS
CIRC {X -108.730,Y 102.264,Z -40.000,A 0.015,B 0.000,C 180.000},{X -95.083,Y 116.070,Z -40.000,A 0.015,B 0.000,C 180.000} C_DIS
CIRC {X -90.133,Y 119.961,Z -40.000,A 0.015,B -0.000,C -180.000},{X -84.867,Y 123.414,Z -40.000,A 0.015,B 0.000,C 180.000} C_DIS
CIRC {X -79.389,Y 126.511,Z -40.000,A 0.015,B -0.000,C -180.000},{X -73.775,Y 129.352,Z -40.000,A 0.015,B 0.000,C 180.000} C_DIS
CIRC {X -70.803,Y 131.996,Z -40.000,A 0.015,B 0.000,C -180.000},{X -69.699,Y 135.817,Z -40.000,A 0.015,B 0.000,C 180.000} C_DIS
LIN {X -69.702,Y 256.213,Z -40.000,A 0.015,B -0.000,C -180.000} C_DIS
CIRC {X -72.011,Y 259.001,Z -40.000,A 0.015,B -0.000,C -180.000},{X -75.181,Y 257.253,Z -40.000,A 0.015,B 0.000,C 180.000} C_DIS
CIRC {X -85.009,Y 238.111,Z -40.000,A 0.015,B 0.000,C -180.000},{X -98.404,Y 221.270,Z -40.000,A 0.015,B 0.000,C 180.000} C_DIS
CIRC {X -114.737,Y 207.283,Z -40.000,A 0.015,B 0.000,C 180.000},{X -133.350,Y 196.514,Z -40.000,A 0.015,B 0.000,C -180.000} C_DIS
CIRC {X -152.995,Y 189.800,Z -40.000,A 0.015,B 0.000,C 180.000},{X -173.598,Y 187.256,Z -40.000,A 0.015,B 0.000,C -180.000} C_DIS
LIN {X -214.895,Y 186.852,Z -40.000,A 0.015,B -0.000,C -180.000} C_DIS
CIRC {X -239.368,Y 189.637,Z -40.000,A 0.015,B 0.000,C 180.000},{X -262.588,Y 197.850,Z -40.000,A 0.015,B -0.000,C 180.000} C_DIS
CIRC {X -274.330,Y 204.406,Z -40.000,A 0.015,B 0.000,C 180.000},{X -285.265,Y 212.233,Z -40.000,A 0.015,B 0.000,C 180.000} C_DIS
CIRC {X -287.807,Y 216.000,Z -40.000,A 0.015,B 0.000,C -180.000},{X -287.777,Y 220.545,Z -40.000,A 0.015,B 0.000,C 180.000} C_DIS
CIRC {X -287.604,Y 225.044,Z -40.000,A 0.015,B 0.000,C 180.000},{X -289.756,Y 228.998,Z -40.000,A 0.015,B 0.000,C 180.000} C_DIS
CIRC {X -292.008,Y 231.406,Z -40.000,A 0.015,B -0.000,C -180.000},{X -294.186,Y 233.879,Z -40.000,A 0.015,B 0.000,C 180.000} C_DIS
CIRC {X -299.545,Y 240.885,Z -40.000,A 0.015,B 0.000,C 180.000},{X -304.113,Y 248.430,Z -40.000,A 0.015,B 0.000,C 180.000} C_DIS
CIRC {X -307.926,Y 256.379,Z -40.000,A 0.015,B 0.000,C 180.000},{X -311.045,Y 264.624,Z -40.000,A 0.015,B -0.000,C 180.000} C_DIS
CIRC {X -313.149,Y 267.498,Z -40.000,A 0.015,B 0.000,C -180.000},{X -316.537,Y 268.595,Z -40.000,A 0.015,B 0.000,C 180.000} C_DIS
LIN {X -329.326,Y 268.594,Z -40.000,A 0.015,B 0.000,C 180.000} C_DIS
CIRC {X -332.050,Y 267.466,Z -40.000,A 0.015,B 0.000,C 180.000},{X -333.179,Y 264.741,Z -40.000,A 0.015,B 0.000,C -180.000} C_DIS
LIN {X -333.175,Y 129.659,Z -40.000,A 0.015,B 0.000,C 180.000} C_DIS
CIRC {X -332.038,Y 125.850,Z -40.000,A 0.015,B 0.000,C 180.000},{X -329.001,Y 123.287,Z -40.000,A 0.015,B 0.000,C -180.000} C_DIS
CIRC {X -321.926,Y 119.980,Z -40.000,A 0.015,B -0.000,C 180.000},{X -315.034,Y 116.307,Z -40.000,A 0.015,B 0.000,C 180.000} C_DIS
CIRC {X -308.458,Y 112.079,Z -40.000,A 0.015,B 0.000,C 180.000},{X -302.390,Y 107.147,Z -40.000,A 0.015,B 0.000,C -180.000} C_DIS
CIRC {X -296.345,Y 101.267,Z -40.000,A 0.015,B 0.000,C 180.000},{X -290.706,Y 94.996,Z -40.000,A 0.015,B 0.000,C 180.000} C_DIS
CIRC {X -285.568,Y 88.304,Z -40.000,A 0.015,B 0.000,C -180.000},{X -281.037,Y 81.187,Z -40.000,A 0.015,B 0.000,C -180.000} C_DIS
LIN {X -263.183,Y 49.543,Z -40.000,A 0.015,B 0.000,C 180.000} C_DIS
CIRC {X -262.368,Y 48.036,Z -40.000,A 0.015,B 0.000,C 180.000},{X -261.636,Y 46.488,Z -40.000,A 0.015,B -0.000,C -180.000} C_DIS
CIRC {X -260.941,Y 44.923,Z -40.000,A 0.015,B 0.000,C -180.000},{X -260.233,Y 43.365,Z -40.000,A 0.015,B 0.000,C -180.000} C_DIS
CIRC {X -257.685,Y 40.433,Z -40.000,A 0.015,B 0.000,C 180.000},{X -253.958,Y 39.341,Z -40.000,A 0.015,B 0.000,C 180.000} C_DIS
LIN {X -139.546,Y 39.341,Z -40.000,A 0.015,B -0.000,C -180.000} C_DIS
CIRC {X -135.803,Y 40.443,Z -40.000,A 0.015,B 0.000,C 180.000},{X -133.254,Y 43.397,Z -40.000,A 0.015,B 0.000,C -180.000} C_DIS
CIRC {X -132.506,Y 45.063,Z -40.000,A 0.015,B 0.000,C 180.000},{X -131.768,Y 46.734,Z -40.000,A 0.015,B 0.000,C -180.000} C_DIS
CIRC {X -130.990,Y 48.386,Z -40.000,A 0.015,B 0.000,C -180.000},{X -130.120,Y 49.993,Z -40.000,A 0.015,B 0.000,C 180.000} C_DIS
LIN {X -109.705,Y 84.933,Z -40.000,A 0.015,B 0.000,C -180.000} C_DIS
CIRC {X -97.457,Y 101.199,Z -40.000,A 0.015,B 0.000,C 180.000},{X -81.905,Y 114.341,Z -40.000,A 0.015,B 0.000,C 180.000} C_DIS
CIRC {X -77.724,Y 116.921,Z -40.000,A 0.015,B 0.000,C 180.000},{X -73.364,Y 119.187,Z -40.000,A 0.015,B -0.000,C 180.000} C_DIS
CIRC {X -68.917,Y 121.268,Z -40.000,A 0.015,B 0.000,C 180.000},{X -64.449,Y 123.305,Z -40.000,A 0.015,B 0.000,C -180.000} C_DIS
CIRC {X -61.454,Y 125.879,Z -40.000,A 0.015,B -0.000,C 180.000},{X -60.336,Y 129.667,Z -40.000,A 0.015,B 0.000,C 180.000} C_DIS
LIN {X -60.339,Y 264.748,Z -40.000,A 0.015,B 0.000,C 180.000} C_DIS
CIRC {X -61.468,Y 267.472,Z -40.000,A 0.015,B -0.000,C 180.000},{X -64.192,Y 268.601,Z -40.000,A 0.015,B -0.000,C 180.000} C_DIS
LIN {X -76.973,Y 268.600,Z -40.000,A 0.015,B 0.000,C -180.000} C_DIS
CIRC {X -80.362,Y 267.504,Z -40.000,A 0.015,B -0.000,C 180.000},{X -82.465,Y 264.630,Z -40.000,A 0.015,B -0.000,C 180.000} C_DIS
CIRC {X -91.113,Y 245.709,Z -40.000,A 0.015,B 0.000,C 180.000},{X -103.677,Y 229.128,Z -40.000,A 0.015,B 0.000,C -180.000} C_DIS
CIRC {X -119.328,Y 215.472,Z -40.000,A 0.015,B 0.000,C -180.000},{X -137.275,Y 205.015,Z -40.000,A 0.015,B -0.000,C -180.000} C_DIS
CIRC {X -155.984,Y 198.673,Z -40.000,A 0.015,B 0.000,C 180.000},{X -175.608,Y 196.401,Z -40.000,A 0.015,B -0.000,C 180.000} C_DIS
LIN {X -214.895,Y 196.215,Z -40.000,A 0.015,B 0.000,C -180.000} C_DIS
CIRC {X -237.362,Y 198.783,Z -40.000,A 0.015,B 0.000,C 180.000},{X -258.670,Y 206.353,Z -40.000,A 0.015,B 0.000,C -180.000} C_DIS
CIRC {X -275.203,Y 216.317,Z -40.000,A 0.015,B 0.000,C -180.000},{X -289.756,Y 228.998,Z -40.000,A 0.015,B 0.000,C -180.000} C_DIS
CIRC {X -291.843,Y 233.173,Z -40.000,A 0.015,B 0.000,C 180.000},{X -291.178,Y 237.792,Z -40.000,A 0.015,B 0.000,C -180.000} C_DIS
CIRC {X -290.326,Y 242.322,Z -40.000,A 0.015,B 0.000,C -180.000},{X -291.838,Y 246.676,Z -40.000,A 0.015,B 0.000,C 180.000} C_DIS
CIRC {X -299.088,Y 259.760,Z -40.000,A 0.015,B 0.000,C 180.000},{X -303.917,Y 273.916,Z -40.000,A 0.015,B -0.000,C 180.000} C_DIS
CIRC {X -305.794,Y 276.827,Z -40.000,A 0.015,B 0.000,C -180.000},{X -309.068,Y 277.957,Z -40.000,A 0.015,B 0.000,C 180.000} C_DIS
LIN {X -338.689,Y 277.957,Z -40.000,A 0.015,B 0.000,C 180.000} C_DIS
CIRC {X -341.413,Y 276.828,Z -40.000,A 0.015,B 0.000,C -180.000},{X -342.541,Y 274.104,Z -40.000,A 0.015,B 0.000,C 180.000} C_DIS
LIN {X -342.537,Y 123.027,Z -40.000,A 0.015,B -0.000,C 180.000} C_DIS
CIRC {X -341.448,Y 119.497,Z -40.000,A 0.015,B -0.000,C 180.000},{X -338.560,Y 117.193,Z -40.000,A 0.015,B 0.000,C 180.000} C_DIS
CIRC {X -329.902,Y 113.433,Z -40.000,A 0.015,B -0.000,C 180.000},{X -321.530,Y 109.070,Z -40.000,A 0.015,B 0.000,C -180.000} C_DIS
CIRC {X -313.582,Y 103.961,Z -40.000,A 0.015,B -0.000,C -180.000},{X -306.251,Y 98.001,Z -40.000,A 0.015,B -0.000,C 180.000} C_DIS
CIRC {X -295.371,Y 86.258,Z -40.000,A 0.015,B 0.000,C 180.000},{X -286.647,Y 72.835,Z -40.000,A 0.015,B 0.000,C -180.000} C_DIS
LIN {X -271.162,Y 44.945,Z -40.000,A 0.015,B -0.000,C 180.000} C_DIS
CIRC {X -269.796,Y 42.332,Z -40.000,A 0.015,B 0.000,C -180.000},{X -268.649,Y 39.615,Z -40.000,A 0.015,B 0.000,C -180.000} C_DIS
CIRC {X -267.593,Y 36.865,Z -40.000,A 0.015,B -0.000,C 180.000},{X -266.494,Y 34.131,Z -40.000,A 0.015,B 0.000,C -180.000} C_DIS
CIRC {X -264.024,Y 31.112,Z -40.000,A 0.015,B 0.000,C 180.000},{X -260.292,Y 29.978,Z -40.000,A 0.015,B 0.000,C 180.000} C_DIS
LIN {X -133.153,Y 29.978,Z -40.000,A 0.015,B 0.000,C -180.000} C_DIS
CIRC {X -129.518,Y 31.074,Z -40.000,A 0.015,B 0.000,C 180.000},{X -127.095,Y 33.996,Z -40.000,A 0.015,B 0.000,C 180.000} C_DIS
CIRC {X -125.918,Y 36.871,Z -40.000,A 0.015,B 0.000,C -180.000},{X -124.801,Y 39.769,Z -40.000,A 0.015,B 0.000,C 180.000} C_DIS
CIRC {X -123.594,Y 42.634,Z -40.000,A 0.015,B 0.000,C -180.000},{X -122.152,Y 45.388,Z -40.000,A 0.015,B 0.000,C 180.000} C_DIS
LIN {X -103.086,Y 78.378,Z -40.000,A 0.015,B 0.000,C -180.000} C_DIS
CIRC {X -91.510,Y 93.983,Z -40.000,A 0.015,B 0.000,C -180.000},{X -76.698,Y 106.559,Z -40.000,A 0.015,B 0.000,C 180.000} C_DIS
CIRC {X -71.529,Y 109.715,Z -40.000,A 0.015,B 0.000,C 180.000},{X -66.116,Y 112.429,Z -40.000,A 0.015,B 0.000,C -180.000} C_DIS
CIRC {X -60.570,Y 114.850,Z -40.000,A 0.015,B 0.000,C 180.000},{X -54.970,Y 117.143,Z -40.000,A 0.015,B -0.000,C -180.000} C_DIS
CIRC {X -52.067,Y 119.469,Z -40.000,A 0.015,B 0.000,C -180.000},{X -50.973,Y 123.026,Z -40.000,A 0.015,B 0.000,C 180.000} C_DIS
LIN {X -50.977,Y 274.111,Z -40.000,A 0.015,B 0.000,C 180.000} C_DIS
CIRC {X -52.106,Y 276.835,Z -40.000,A 0.015,B 0.000,C -180.000},{X -54.830,Y 277.963,Z -40.000,A 0.015,B 0.000,C -180.000} C_DIS
LIN {X -84.491,Y 277.963,Z -40.000,A 0.015,B 0.000,C -180.000} C_DIS
CIRC {X -87.751,Y 276.829,Z -40.000,A 0.015,B 0.000,C 180.000},{X -89.604,Y 273.919,Z -40.000,A 0.015,B 0.000,C 180.000} C_DIS
CIRC {X -96.331,Y 255.347,Z -40.000,A 0.015,B 0.000,C -180.000},{X -107.119,Y 238.799,Z -40.000,A 0.015,B 0.000,C -180.000} C_DIS
CIRC {X -121.340,Y 225.102,Z -40.000,A 0.015,B 0.000,C 180.000},{X -138.235,Y 214.884,Z -40.000,A 0.015,B -0.000,C 180.000} C_DIS
CIRC {X -147.910,Y 210.979,Z -40.000,A 0.015,B 0.000,C -180.000},{X -157.920,Y 208.039,Z -40.000,A 0.015,B 0.000,C 180.000} C_DIS
CIRC {X -168.196,Y 206.195,Z -40.000,A 0.015,B -0.000,C 180.000},{X -178.617,Y 205.578,Z -40.000,A 0.015,B 0.000,C -180.000} C_DIS
LIN {X -217.249,Y 205.684,Z -40.000,A 0.015,B -0.000,C -180.000} C_DIS
CIRC {X -236.552,Y 208.014,Z -40.000,A 0.015,B 0.000,C -180.000},{X -254.821,Y 214.671,Z -40.000,A 0.015,B 0.000,C -180.000} C_DIS
CIRC {X -271.558,Y 225.237,Z -40.000,A 0.015,B 0.000,C 180.000},{X -285.889,Y 238.891,Z -40.000,A 0.015,B -0.000,C 180.000} C_DIS
CIRC {X -288.976,Y 242.697,Z -40.000,A 0.015,B 0.000,C 180.000},{X -291.838,Y 246.676,Z -40.000,A 0.015,B 0.000,C 180.000} C_DIS
CIRC {X -293.117,Y 250.967,Z -40.000,A 0.015,B -0.000,C -180.000},{X -291.708,Y 255.217,Z -40.000,A 0.015,B 0.000,C -180.000} C_DIS
CIRC {X -290.118,Y 259.336,Z -40.000,A 0.015,B 0.000,C 180.000},{X -290.756,Y 263.705,Z -40.000,A 0.015,B 0.000,C 180.000} C_DIS
CIRC {X -291.592,Y 265.755,Z -40.000,A 0.015,B 0.000,C -180.000},{X -292.369,Y 267.829,Z -40.000,A 0.015,B -0.000,C 180.000} C_DIS
CIRC {X -294.262,Y 273.684,Z -40.000,A 0.015,B 0.000,C -180.000},{X -295.789,Y 279.645,Z -40.000,A 0.015,B -0.000,C -180.000} C_DIS
CIRC {X -295.977,Y 280.553,Z -40.000,A 0.015,B 0.000,C 180.000},{X -296.136,Y 281.468,Z -40.000,A 0.015,B 0.000,C -180.000} C_DIS
CIRC {X -296.296,Y 282.382,Z -40.000,A 0.015,B 0.000,C 180.000},{X -296.484,Y 283.291,Z -40.000,A 0.015,B -0.000,C 180.000} C_DIS
CIRC {X -298.291,Y 286.189,Z -40.000,A 0.015,B 0.000,C -180.000},{X -301.513,Y 287.320,Z -40.000,A 0.015,B 0.000,C -180.000} C_DIS
LIN {X -348.051,Y 287.319,Z -40.000,A 0.015,B -0.000,C -180.000} C_DIS
CIRC {X -350.776,Y 286.190,Z -40.000,A 0.015,B 0.000,C 180.000},{X -351.904,Y 283.466,Z -40.000,A 0.015,B -0.000,C 180.000} C_DIS
LIN {X -351.900,Y 115.525,Z -40.000,A 0.015,B 0.000,C 180.000} C_DIS
CIRC {X -350.811,Y 112.325,Z -40.000,A 0.015,B -0.000,C 180.000},{X -347.997,Y 110.451,Z -40.000,A 0.015,B 0.000,C 180.000} C_DIS
CIRC {X -321.730,Y 98.251,Z -40.000,A 0.015,B -0.000,C -180.000},{X -301.244,Y 77.778,Z -40.000,A 0.015,B 0.000,C 180.000} C_DIS
CIRC {X -286.180,Y 53.511,Z -40.000,A 0.015,B 0.000,C 180.000},{X -273.872,Y 27.736,Z -40.000,A 0.015,B 0.000,C -180.000} C_DIS
CIRC {X -273.570,Y 26.951,Z -40.000,A 0.015,B -0.000,C -180.000},{X -273.305,Y 26.152,Z -40.000,A 0.015,B 0.000,C 180.000} C_DIS
CIRC {X -273.051,Y 25.349,Z -40.000,A 0.015,B 0.000,C -180.000},{X -272.785,Y 24.551,Z -40.000,A 0.015,B 0.000,C 180.000} C_DIS
CIRC {X -270.663,Y 21.700,Z -40.000,A 0.015,B 0.000,C 180.000},{X -267.279,Y 20.615,Z -40.000,A 0.015,B -0.000,C -180.000} C_DIS
LIN {X -126.310,Y 20.615,Z -40.000,A 0.015,B 0.000,C 180.000} C_DIS
CIRC {X -122.890,Y 21.699,Z -40.000,A 0.015,B -0.000,C -180.000},{X -120.719,Y 24.555,Z -40.000,A 0.015,B 0.000,C 180.000} C_DIS
CIRC {X -115.565,Y 37.155,Z -40.000,A 0.015,B 0.000,C -180.000},{X -109.294,Y 49.237,Z -40.000,A 0.015,B -0.000,C 180.000} C_DIS
LIN {X -96.034,Y 72.181,Z -40.000,A 0.015,B 0.000,C 180.000} C_DIS
CIRC {X -86.526,Y 85.340,Z -40.000,A 0.015,B -0.000,C -180.000},{X -74.556,Y 96.308,Z -40.000,A 0.015,B 0.000,C -180.000} C_DIS
CIRC {X -60.698,Y 104.741,Z -40.000,A 0.015,B 0.000,C -180.000},{X -45.516,Y 110.454,Z -40.000,A 0.015,B 0.000,C 180.000} C_DIS
CIRC {X -42.698,Y 112.351,Z -40.000,A 0.015,B 0.000,C 180.000},{X -41.610,Y 115.569,Z -40.000,A 0.015,B 0.000,C -180.000} C_DIS
LIN {X -41.615,Y 283.473,Z -40.000,A 0.015,B 0.000,C -180.000} C_DIS
CIRC {X -42.743,Y 286.198,Z -40.000,A 0.015,B -0.000,C 180.000},{X -45.468,Y 287.326,Z -40.000,A 0.015,B 0.000,C -180.000} C_DIS
LIN {X -91.941,Y 287.325,Z -40.000,A 0.015,B -0.000,C -180.000} C_DIS
CIRC {X -95.165,Y 286.204,Z -40.000,A 0.015,B -0.000,C -180.000},{X -96.999,Y 283.324,Z -40.000,A 0.015,B 0.000,C 180.000} C_DIS
LIN {X -99.674,Y 271.837,Z -40.000,A 0.015,B 0.000,C 180.000} C_DIS
CIRC {X -101.394,Y 266.181,Z -40.000,A 0.015,B 0.000,C 180.000},{X -103.886,Y 260.820,Z -40.000,A 0.015,B 0.000,C 180.000} C_DIS
CIRC {X -117.367,Y 242.306,Z -40.000,A 0.015,B 0.000,C -180.000},{X -134.990,Y 227.682,Z -40.000,A 0.015,B 0.000,C -180.000} C_DIS
CIRC {X -155.892,Y 218.191,Z -40.000,A 0.015,B 0.000,C -180.000},{X -178.617,Y 214.940,Z -40.000,A 0.015,B 0.000,C -180.000} C_DIS
LIN {X -221.198,Y 215.566,Z -40.000,A 0.015,B 0.000,C -180.000} C_DIS
CIRC {X -242.387,Y 219.405,Z -40.000,A 0.015,B 0.000,C 180.000},{X -261.499,Y 229.327,Z -40.000,A 0.015,B 0.000,C 180.000} C_DIS
CIRC {X -268.930,Y 235.171,Z -40.000,A 0.015,B 0.000,C 180.000},{X -275.899,Y 241.557,Z -40.000,A 0.015,B 0.000,C -180.000} C_DIS
CIRC {X -282.141,Y 248.680,Z -40.000,A 0.015,B -0.000,C -180.000},{X -287.304,Y 256.619,Z -40.000,A 0.015,B 0.000,C -180.000} C_DIS
CIRC {X -289.122,Y 260.118,Z -40.000,A 0.015,B 0.000,C 180.000},{X -290.756,Y 263.705,Z -40.000,A 0.015,B 0.000,C 180.000} C_DIS
CIRC {X -291.220,Y 268.093,Z -40.000,A 0.015,B 0.000,C 180.000},{X -289.152,Y 271.990,Z -40.000,A 0.015,B -0.000,C 180.000} C_DIS
CIRC {X -286.925,Y 275.728,Z -40.000,A 0.015,B 0.000,C -180.000},{X -286.732,Y 280.075,Z -40.000,A 0.015,B 0.000,C 180.000} C_DIS
CIRC {X -287.891,Y 286.458,Z -40.000,A 0.015,B 0.000,C -180.000},{X -288.757,Y 292.887,Z -40.000,A 0.015,B -0.000,C 180.000} C_DIS
CIRC {X -290.154,Y 295.595,Z -40.000,A 0.015,B 0.000,C -180.000},{X -293.001,Y 296.683,Z -40.000,A 0.015,B 0.000,C 180.000} C_DIS
LIN {X -357.414,Y 296.681,Z -40.000,A 0.015,B 0.000,C -180.000} C_DIS
CIRC {X -360.139,Y 295.553,Z -40.000,A 0.015,B -0.000,C 180.000},{X -361.267,Y 292.828,Z -40.000,A 0.015,B 0.000,C -180.000} C_DIS
LIN {X -361.262,Y 107.566,Z -40.000,A 0.015,B 0.000,C 180.000} C_DIS
CIRC {X -360.165,Y 104.514,Z -40.000,A 0.015,B -0.000,C -180.000},{X -357.376,Y 102.859,Z -40.000,A 0.015,B 0.000,C -180.000} C_DIS
CIRC {X -353.906,Y 102.202,Z -40.000,A 0.015,B -0.000,C 180.000},{X -350.433,Y 101.568,Z -40.000,A 0.015,B -0.000,C -180.000} C_DIS
CIRC {X -346.993,Y 100.742,Z -40.000,A 0.015,B 0.000,C -180.000},{X -343.674,Y 99.521,Z -40.000,A 0.015,B -0.000,C -180.000} C_DIS
CIRC {X -332.369,Y 93.684,Z -40.000,A 0.015,B 0.000,C -180.000},{X -321.925,Y 86.418,Z -40.000,A 0.015,B 0.000,C 180.000} C_DIS
CIRC {X -312.745,Y 77.568,Z -40.000,A 0.015,B 0.000,C -180.000},{X -305.374,Y 67.163,Z -40.000,A 0.015,B 0.000,C -180.000} C_DIS
LIN {X -290.629,Y 42.137,Z -40.000,A 0.015,B 0.000,C -180.000} C_DIS
CIRC {X -284.146,Y 29.087,Z -40.000,A 0.015,B 0.000,C -180.000},{X -279.855,Y 15.163,Z -40.000,A 0.015,B 0.000,C -180.000} C_DIS
CIRC {X -278.108,Y 12.351,Z -40.000,A 0.015,B 0.000,C 180.000},{X -274.985,Y 11.253,Z -40.000,A 0.015,B 0.000,C -180.000} C_DIS
LIN {X -118.591,Y 11.253,Z -40.000,A 0.015,B 0.000,C -180.000} C_DIS
CIRC {X -115.396,Y 12.384,Z -40.000,A 0.015,B -0.000,C 180.000},{X -113.624,Y 15.274,Z -40.000,A 0.015,B 0.000,C -180.000} C_DIS
CIRC {X -112.306,Y 20.672,Z -40.000,A 0.015,B -0.000,C 180.000},{X -110.669,Y 25.982,Z -40.000,A 0.015,B 0.000,C -180.000} C_DIS
CIRC {X -108.619,Y 31.151,Z -40.000,A 0.015,B 0.000,C -180.000},{X -106.074,Y 36.096,Z -40.000,A 0.015,B 0.000,C 180.000} C_DIS
LIN {X -84.464,Y 72.658,Z -40.000,A 0.015,B 0.000,C 180.000} C_DIS
CIRC {X -75.235,Y 82.926,Z -40.000,A 0.015,B 0.000,C 180.000},{X -64.590,Y 91.716,Z -40.000,A 0.015,B 0.000,C -180.000} C_DIS
CIRC {X -52.482,Y 98.442,Z -40.000,A 0.015,B -0.000,C 180.000},{X -39.207,Y 102.392,Z -40.000,A 0.015,B 0.000,C 180.000} C_DIS
CIRC {X -38.461,Y 102.516,Z -40.000,A 0.015,B 0.000,C 180.000},{X -37.711,Y 102.616,Z -40.000,A 0.015,B 0.000,C 180.000} C_DIS
CIRC {X -36.962,Y 102.717,Z -40.000,A 0.015,B 0.000,C -180.000},{X -36.216,Y 102.841,Z -40.000,A 0.015,B 0.000,C -180.000} C_DIS
CIRC {X -33.370,Y 104.500,Z -40.000,A 0.015,B -0.000,C 180.000},{X -32.247,Y 107.598,Z -40.000,A 0.015,B 0.000,C -180.000} C_DIS
LIN {X -32.252,Y 292.836,Z -40.000,A 0.015,B 0.000,C -180.000} C_DIS
CIRC {X -33.381,Y 295.561,Z -40.000,A 0.015,B 0.000,C -180.000},{X -36.105,Y 296.689,Z -40.000,A 0.015,B -0.000,C -180.000} C_DIS
LIN {X -100.545,Y 296.688,Z -40.000,A 0.015,B 0.000,C 180.000} C_DIS
CIRC {X -103.376,Y 295.599,Z -40.000,A 0.015,B -0.000,C -180.000},{X -104.750,Y 292.896,Z -40.000,A 0.015,B -0.000,C -180.000} C_DIS
CIRC {X -106.471,Y 282.433,Z -40.000,A 0.015,B 0.000,C 180.000},{X -109.434,Y 272.253,Z -40.000,A 0.015,B 0.000,C -180.000} C_DIS
CIRC {X -113.756,Y 262.558,Z -40.000,A 0.015,B 0.000,C -180.000},{X -119.498,Y 253.631,Z -40.000,A 0.015,B 0.000,C 180.000} C_DIS
CIRC {X -125.716,Y 246.484,Z -40.000,A 0.015,B 0.000,C 180.000},{X -132.850,Y 240.252,Z -40.000,A 0.015,B 0.000,C 180.000} C_DIS
CIRC {X -140.686,Y 234.943,Z -40.000,A 0.015,B 0.000,C -180.000},{X -149.051,Y 230.515,Z -40.000,A 0.015,B 0.000,C -180.000} C_DIS
CIRC {X -154.628,Y 228.319,Z -40.000,A 0.015,B 0.000,C -180.000},{X -160.421,Y 226.776,Z -40.000,A 0.015,B 0.000,C 180.000} C_DIS
CIRC {X -166.302,Y 225.666,Z -40.000,A 0.015,B 0.000,C 180.000},{X -172.216,Y 224.746,Z -40.000,A 0.015,B 0.000,C -180.000} C_DIS
LIN {X -214.895,Y 224.303,Z -40.000,A 0.015,B -0.000,C -180.000} C_DIS
CIRC {X -235.155,Y 227.223,Z -40.000,A 0.015,B 0.000,C -180.000},{X -253.765,Y 235.746,Z -40.000,A 0.015,B 0.000,C -180.000} C_DIS
CIRC {X -269.433,Y 248.834,Z -40.000,A 0.015,B 0.000,C 180.000},{X -281.433,Y 265.350,Z -40.000,A 0.015,B 0.000,C 180.000} C_DIS
CIRC {X -284.436,Y 271.869,Z -40.000,A 0.015,B 0.000,C 180.000},{X -286.455,Y 278.757,Z -40.000,A 0.015,B 0.000,C -180.000} C_DIS
CIRC {X -286.595,Y 279.415,Z -40.000,A 0.015,B 0.000,C 180.000},{X -286.732,Y 280.075,Z -40.000,A 0.015,B -0.000,C 180.000} C_DIS
CIRC {X -286.322,Y 284.447,Z -40.000,A 0.015,B 0.000,C -180.000},{X -283.544,Y 287.847,Z -40.000,A 0.015,B -0.000,C 180.000} C_DIS
CIRC {X -280.652,Y 291.079,Z -40.000,A 0.015,B 0.000,C -180.000},{X -279.673,Y 295.303,Z -40.000,A 0.015,B 0.000,C -180.000} C_DIS
CIRC {X -279.654,Y 298.860,Z -40.000,A 0.015,B 0.000,C 180.000},{X -279.431,Y 302.410,Z -40.000,A 0.015,B 0.000,C 180.000} C_DIS
CIRC {X -280.287,Y 304.960,Z -40.000,A 0.015,B 0.000,C 180.000},{X -282.747,Y 306.046,Z -40.000,A 0.015,B 0.000,C 180.000} C_DIS
LIN {X -366.777,Y 306.044,Z -40.000,A 0.015,B 0.000,C -180.000} C_DIS
CIRC {X -369.502,Y 304.915,Z -40.000,A 0.015,B 0.000,C 180.000},{X -370.630,Y 302.191,Z -40.000,A 0.015,B 0.000,C -180.000} C_DIS
LIN {X -370.624,Y 98.537,Z -40.000,A 0.015,B 0.000,C 180.000} C_DIS
CIRC {X -369.544,Y 95.832,Z -40.000,A 0.015,B 0.000,C -180.000},{X -366.896,Y 94.618,Z -40.000,A 0.015,B 0.000,C 180.000} C_DIS
CIRC {X -344.508,Y 89.557,Z -40.000,A 0.015,B 0.000,C 180.000},{X -325.151,Y 77.224,Z -40.000,A 0.015,B 0.000,C 180.000} C_DIS
CIRC {X -322.594,Y 74.682,Z -40.000,A 0.015,B -0.000,C -180.000},{X -320.272,Y 71.923,Z -40.000,A 0.015,B 0.000,C 180.000} C_DIS
CIRC {X -318.086,Y 69.060,Z -40.000,A 0.015,B -0.000,C -180.000},{X -315.920,Y 66.183,Z -40.000,A 0.015,B 0.000,C -180.000} C_DIS
LIN {X -295.346,Y 31.009,Z -40.000,A 0.015,B 0.000,C 180.000} C_DIS
CIRC {X -292.386,Y 25.057,Z -40.000,A 0.015,B 0.000,C -180.000},{X -290.178,Y 18.787,Z -40.000,A 0.015,B 0.000,C -180.000} C_DIS
CIRC {X -288.655,Y 12.321,Z -40.000,A 0.015,B -0.000,C -180.000},{X -287.733,Y 5.744,Z -40.000,A 0.015,B 0.000,C 180.000} C_DIS
CIRC {X -286.363,Y 2.998,Z -40.000,A 0.015,B -0.000,C -180.000},{X -283.502,Y 1.890,Z -40.000,A 0.015,B 0.000,C 180.000} C_DIS
LIN {X -110.045,Y 1.890,Z -40.000,A 0.015,B 0.000,C 180.000} C_DIS
CIRC {X -107.132,Y 3.017,Z -40.000,A 0.015,B 0.000,C 180.000},{X -105.735,Y 5.811,Z -40.000,A 0.015,B 0.000,C -180.000} C_DIS
CIRC {X -104.790,Y 12.478,Z -40.000,A 0.015,B 0.000,C -180.000},{X -103.232,Y 19.030,Z -40.000,A 0.015,B 0.000,C 180.000} C_DIS
CIRC {X -100.978,Y 25.381,Z -40.000,A 0.015,B -0.000,C 180.000},{X -97.968,Y 31.412,Z -40.000,A 0.015,B -0.000,C 180.000} C_DIS
LIN {X -77.056,Y 66.933,Z -40.000,A 0.015,B -0.000,C 180.000} C_DIS
CIRC {X -68.999,Y 75.984,Z -40.000,A 0.015,B 0.000,C 180.000},{X -59.768,Y 83.835,Z -40.000,A 0.015,B 0.000,C -180.000} C_DIS
CIRC {X -49.219,Y 89.898,Z -40.000,A 0.015,B 0.000,C 180.000},{X -37.573,Y 93.424,Z -40.000,A 0.015,B -0.000,C 180.000} C_DIS
CIRC {X -34.866,Y 93.856,Z -40.000,A 0.015,B 0.000,C 180.000},{X -32.143,Y 94.168,Z -40.000,A 0.015,B 0.000,C -180.000} C_DIS
CIRC {X -29.412,Y 94.395,Z -40.000,A 0.015,B -0.000,C 180.000},{X -26.677,Y 94.570,Z -40.000,A 0.015,B -0.000,C -180.000} C_DIS
CIRC {X -23.983,Y 95.818,Z -40.000,A 0.015,B 0.000,C 180.000},{X -22.884,Y 98.577,Z -40.000,A 0.015,B 0.000,C 180.000} C_DIS
LIN {X -22.890,Y 302.199,Z -40.000,A 0.015,B 0.000,C 180.000} C_DIS
CIRC {X -24.019,Y 304.924,Z -40.000,A 0.015,B -0.000,C 180.000},{X -26.743,Y 306.052,Z -40.000,A 0.015,B 0.000,C 180.000} C_DIS
LIN {X -110.801,Y 306.050,Z -40.000,A 0.015,B -0.000,C -180.000} C_DIS
CIRC {X -113.247,Y 304.956,Z -40.000,A 0.015,B 0.000,C -180.000},{X -114.062,Y 302.404,Z -40.000,A 0.015,B 0.000,C -180.000} C_DIS
CIRC {X -115.318,Y 282.600,Z -40.000,A 0.015,B 0.000,C -180.000},{X -123.282,Y 264.425,Z -40.000,A 0.015,B 0.000,C 180.000} C_DIS
CIRC {X -136.370,Y 249.664,Z -40.000,A 0.015,B 0.000,C -180.000},{X -152.976,Y 239.015,Z -40.000,A 0.015,B 0.000,C 180.000} C_DIS
CIRC {X -157.919,Y 237.084,Z -40.000,A 0.015,B 0.000,C 180.000},{X -163.057,Y 235.760,Z -40.000,A 0.015,B 0.000,C 180.000} C_DIS
CIRC {X -168.270,Y 234.820,Z -40.000,A 0.015,B 0.000,C 180.000},{X -173.506,Y 234.019,Z -40.000,A 0.015,B 0.000,C -180.000} C_DIS
LIN {X -214.895,Y 233.665,Z -40.000,A 0.015,B 0.000,C -180.000} C_DIS
CIRC {X -240.661,Y 238.907,Z -40.000,A 0.015,B 0.000,C -180.000},{X -262.332,Y 253.797,Z -40.000,A 0.015,B 0.000,C 180.000} C_DIS
CIRC {X -274.911,Y 272.917,Z -40.000,A 0.015,B 0.000,C -180.000},{X -279.673,Y 295.303,Z -40.000,A 0.015,B -0.000,C -180.000} C_DIS
CIRC {X -278.421,Y 299.461,Z -40.000,A 0.015,B 0.000,C 180.000},{X -274.955,Y 302.077,Z -40.000,A 0.015,B 0.000,C -180.000} C_DIS
CIRC {X -271.410,Y 304.463,Z -40.000,A 0.015,B 0.000,C -180.000},{X -269.536,Y 308.304,Z -40.000,A 0.015,B -0.000,C 180.000} C_DIS
CIRC {X -269.253,Y 309.843,Z -40.000,A 0.015,B 0.000,C -180.000},{X -269.001,Y 311.388,Z -40.000,A 0.015,B -0.000,C -180.000} C_DIS
CIRC {X -269.735,Y 313.951,Z -40.000,A 0.015,B 0.000,C 180.000},{X -272.158,Y 315.064,Z -40.000,A 0.015,B -0.000,C 180.000} C_DIS
LIN {X -375.795,Y 315.061,Z -40.000,A 0.015,B 0.000,C 180.000} C_DIS
CIRC {X -378.520,Y 313.933,Z -40.000,A 0.015,B -0.000,C 180.000},{X -379.648,Y 311.208,Z -40.000,A 0.015,B 0.000,C -180.000} C_DIS
LIN {X -379.642,Y 88.701,Z -40.000,A 0.015,B -0.000,C -180.000} C_DIS
CIRC {X -378.568,Y 86.272,Z -40.000,A 0.015,B 0.000,C 180.000},{X -376.048,Y 85.433,Z -40.000,A 0.015,B 0.000,C -180.000} C_DIS
CIRC {X -355.323,Y 83.747,Z -40.000,A 0.015,B 0.000,C 180.000},{X -336.456,Y 75.008,Z -40.000,A 0.015,B 0.000,C -180.000} C_DIS
CIRC {X -332.632,Y 71.949,Z -40.000,A 0.015,B 0.000,C 180.000},{X -329.232,Y 68.426,Z -40.000,A 0.015,B 0.000,C -180.000} C_DIS
CIRC {X -326.128,Y 64.651,Z -40.000,A 0.015,B 0.000,C -180.000},{X -323.141,Y 60.782,Z -40.000,A 0.015,B -0.000,C 180.000} C_DIS
LIN {X -303.159,Y 26.506,Z -40.000,A 0.015,B 0.000,C 180.000} C_DIS
CIRC {X -299.818,Y 19.497,Z -40.000,A 0.015,B 0.000,C -180.000},{X -297.605,Y 12.054,Z -40.000,A 0.015,B -0.000,C 180.000} C_DIS
CIRC {X -296.512,Y 4.371,Z -40.000,A 0.015,B 0.000,C 180.000},{X -296.501,Y -3.389,Z -40.000,A 0.015,B 0.000,C -180.000} C_DIS
CIRC {X -295.567,Y -6.017,Z -40.000,A 0.015,B 0.000,C -180.000},{X -293.010,Y -7.128,Z -40.000,A 0.015,B 0.000,C 180.000} C_DIS
LIN {X -100.416,Y -7.128,Z -40.000,A 0.015,B -0.000,C -180.000} C_DIS
CIRC {X -97.919,Y -6.035,Z -40.000,A 0.015,B 0.000,C 180.000},{X -97.027,Y -3.460,Z -40.000,A 0.015,B 0.000,C 180.000} C_DIS
CIRC {X -95.705,Y 13.546,Z -40.000,A 0.015,B 0.000,C -180.000},{X -89.211,Y 29.319,Z -40.000,A 0.015,B 0.000,C 180.000} C_DIS
LIN {X -72.014,Y 58.299,Z -40.000,A 0.015,B 0.000,C 180.000} C_DIS
CIRC {X -61.995,Y 70.845,Z -40.000,A 0.015,B 0.000,C 180.000},{X -48.719,Y 79.873,Z -40.000,A 0.015,B 0.000,C -180.000} C_DIS
CIRC {X -33.469,Y 84.786,Z -40.000,A 0.015,B -0.000,C 180.000},{X -17.460,Y 85.433,Z -40.000,A 0.015,B 0.000,C 180.000} C_DIS
CIRC {X -14.941,Y 86.271,Z -40.000,A 0.015,B 0.000,C 180.000},{X -13.866,Y 88.700,Z -40.000,A 0.015,B 0.000,C 180.000} C_DIS
LIN {X -13.872,Y 311.217,Z -40.000,A 0.015,B 0.000,C -180.000} C_DIS
CIRC {X -15.001,Y 313.942,Z -40.000,A 0.015,B 0.000,C -180.000},{X -17.725,Y 315.070,Z -40.000,A 0.015,B 0.000,C 180.000} C_DIS
LIN {X -121.355,Y 315.068,Z -40.000,A 0.015,B 0.000,C 180.000} C_DIS
CIRC {X -123.758,Y 313.967,Z -40.000,A 0.015,B 0.000,C 180.000},{X -124.494,Y 311.428,Z -40.000,A 0.015,B 0.000,C 180.000} C_DIS
CIRC {X -123.703,Y 306.386,Z -40.000,A 0.015,B -0.000,C 180.000},{X -122.831,Y 301.356,Z -40.000,A 0.015,B 0.000,C -180.000} C_DIS
CIRC {X -122.437,Y 296.240,Z -40.000,A 0.015,B 0.000,C 180.000},{X -123.098,Y 291.151,Z -40.000,A 0.015,B -0.000,C 180.000} C_DIS
CIRC {X -125.078,Y 283.787,Z -40.000,A 0.015,B 0.000,C -180.000},{X -127.499,Y 276.555,Z -40.000,A 0.015,B 0.000,C -180.000} C_DIS
CIRC {X -130.772,Y 269.638,Z -40.000,A 0.015,B 0.000,C 180.000},{X -135.214,Y 263.407,Z -40.000,A 0.015,B 0.000,C -180.000} C_DIS
CIRC {X -144.164,Y 254.865,Z -40.000,A 0.015,B 0.000,C 180.000},{X -154.645,Y 248.289,Z -40.000,A 0.015,B 0.000,C 180.000} C_DIS
CIRC {X -166.307,Y 244.103,Z -40.000,A 0.015,B 0.000,C 180.000},{X -178.617,Y 242.683,Z -40.000,A 0.015,B -0.000,C -180.000} C_DIS
LIN {X -218.763,Y 242.951,Z -40.000,A 0.015,B -0.000,C -180.000} C_DIS
CIRC {X -230.671,Y 245.620,Z -40.000,A 0.015,B 0.000,C 180.000},{X -241.981,Y 250.204,Z -40.000,A 0.015,B 0.000,C -180.000} C_DIS
CIRC {X -252.170,Y 257.010,Z -40.000,A 0.015,B -0.000,C -180.000},{X -260.421,Y 266.069,Z -40.000,A 0.015,B -0.000,C 180.000} C_DIS
CIRC {X -265.153,Y 273.879,Z -40.000,A 0.015,B 0.000,C 180.000},{X -268.710,Y 282.290,Z -40.000,A 0.015,B 0.000,C -180.000} C_DIS
CIRC {X -270.746,Y 291.218,Z -40.000,A 0.015,B -0.000,C -180.000},{X -270.905,Y 300.374,Z -40.000,A 0.015,B 0.000,C 180.000} C_DIS
CIRC {X -270.569,Y 303.150,Z -40.000,A 0.015,B 0.000,C 180.000},{X -270.043,Y 305.897,Z -40.000,A 0.015,B 0.000,C -180.000} C_DIS
CIRC {X -269.780,Y 307.098,Z -40.000,A 0.015,B -0.000,C -180.000},{X -269.536,Y 308.304,Z -40.000,A 0.015,B 0.000,C -180.000} C_DIS
CIRC {X -267.619,Y 311.889,Z -40.000,A 0.015,B 0.000,C -180.000},{X -264.015,Y 313.771,Z -40.000,A 0.015,B 0.000,C 180.000} C_DIS
CIRC {X -260.363,Y 315.388,Z -40.000,A 0.015,B 0.000,C 180.000},{X -257.837,Y 318.482,Z -40.000,A 0.015,B 0.000,C 180.000} C_DIS
CIRC {X -257.358,Y 319.442,Z -40.000,A 0.015,B 0.000,C -180.000},{X -256.853,Y 320.390,Z -40.000,A 0.015,B 0.000,C 180.000} C_DIS
CIRC {X -256.889,Y 322.643,Z -40.000,A 0.015,B 0.000,C 180.000},{X -258.847,Y 323.760,Z -40.000,A 0.015,B -0.000,C -180.000} C_DIS
LIN {X -384.491,Y 323.757,Z -40.000,A 0.015,B -0.000,C -180.000} C_DIS
CIRC {X -387.215,Y 322.628,Z -40.000,A 0.015,B 0.000,C -180.000},{X -388.344,Y 319.904,Z -40.000,A 0.015,B 0.000,C 180.000} C_DIS
LIN {X -388.337,Y 76.981,Z -40.000,A 0.015,B -0.000,C -180.000} C_DIS
CIRC {X -387.215,Y 74.745,Z -40.000,A 0.015,B 0.000,C 180.000},{X -384.752,Y 74.308,Z -40.000,A 0.015,B -0.000,C -180.000} C_DIS
CIRC {X -382.044,Y 75.170,Z -40.000,A 0.015,B -0.000,C 180.000},{X -379.370,Y 76.131,Z -40.000,A 0.015,B -0.000,C -180.000} C_DIS
CIRC {X -376.628,Y 76.912,Z -40.000,A 0.015,B -0.000,C -180.000},{X -373.792,Y 77.211,Z -40.000,A 0.015,B 0.000,C 180.000} C_DIS
CIRC {X -364.627,Y 76.756,Z -40.000,A 0.015,B 0.000,C -180.000},{X -355.610,Y 75.058,Z -40.000,A 0.015,B 0.000,C -180.000} C_DIS
CIRC {X -347.030,Y 71.677,Z -40.000,A 0.015,B 0.000,C -180.000},{X -339.510,Y 66.340,Z -40.000,A 0.015,B 0.000,C 180.000} C_DIS
CIRC {X -336.511,Y 63.455,Z -40.000,A 0.015,B 0.000,C 180.000},{X -333.679,Y 60.406,Z -40.000,A 0.015,B 0.000,C -180.000} C_DIS
CIRC {X -331.089,Y 57.145,Z -40.000,A 0.015,B 0.000,C 180.000},{X -328.833,Y 53.644,Z -40.000,A 0.015,B 0.000,C 180.000} C_DIS
LIN {X -309.564,Y 19.867,Z -40.000,A 0.015,B 0.000,C -180.000} C_DIS
CIRC {X -307.585,Y 14.623,Z -40.000,A 0.015,B -0.000,C -180.000},{X -305.920,Y 9.272,Z -40.000,A 0.015,B 0.000,C -180.000} C_DIS
CIRC {X -304.875,Y 3.748,Z -40.000,A 0.015,B -0.000,C 180.000},{X -304.781,Y -1.873,Z -40.000,A 0.015,B 0.000,C -180.000} C_DIS
CIRC {X -305.355,Y -7.156,Z -40.000,A 0.015,B -0.000,C 180.000},{X -306.347,Y -12.376,Z -40.000,A 0.015,B 0.000,C 180.000} C_DIS
CIRC {X -305.803,Y -14.762,Z -40.000,A 0.015,B 0.000,C 180.000},{X -303.599,Y -15.823,Z -40.000,A 0.015,B 0.000,C 180.000} C_DIS
LIN {X -89.913,Y -15.823,Z -40.000,A 0.015,B 0.000,C -180.000} C_DIS
CIRC {X -87.708,Y -14.762,Z -40.000,A 0.015,B 0.000,C 180.000},{X -87.165,Y -12.376,Z -40.000,A 0.015,B 0.000,C -180.000} C_DIS
CIRC {X -88.156,Y -6.830,Z -40.000,A 0.015,B 0.000,C -180.000},{X -88.612,Y -1.214,Z -40.000,A 0.015,B 0.000,C 180.000} C_DIS
CIRC {X -88.457,Y 4.421,Z -40.000,A 0.015,B 0.000,C 180.000},{X -87.620,Y 9.997,Z -40.000,A 0.015,B -0.000,C 180.000} C_DIS
CIRC {X -86.899,Y 12.694,Z -40.000,A 0.015,B 0.000,C -180.000},{X -85.906,Y 15.303,Z -40.000,A 0.015,B -0.000,C 180.000} C_DIS
CIRC {X -84.790,Y 17.858,Z -40.000,A 0.015,B 0.000,C 180.000},{X -83.693,Y 20.420,Z -40.000,A 0.015,B -0.000,C 180.000} C_DIS
LIN {X -64.485,Y 53.948,Z -40.000,A 0.015,B 0.000,C 180.000} C_DIS
CIRC {X -57.229,Y 63.407,Z -40.000,A 0.015,B -0.000,C 180.000},{X -47.780,Y 70.675,Z -40.000,A 0.015,B 0.000,C 180.000} C_DIS
CIRC {X -36.854,Y 75.395,Z -40.000,A 0.015,B 0.000,C -180.000},{X -25.128,Y 77.437,Z -40.000,A 0.015,B -0.000,C 180.000} C_DIS
CIRC {X -22.462,Y 77.475,Z -40.000,A 0.015,B -0.000,C -180.000},{X -19.802,Y 77.300,Z -40.000,A 0.015,B 0.000,C -180.000} C_DIS
CIRC {X -17.167,Y 76.893,Z -40.000,A 0.015,B 0.000,C 180.000},{X -14.581,Y 76.242,Z -40.000,A 0.015,B -0.000,C -180.000} C_DIS
CIRC {X -13.116,Y 75.775,Z -40.000,A 0.015,B 0.000,C -180.000},{X -11.666,Y 75.262,Z -40.000,A 0.015,B 0.000,C 180.000} C_DIS
CIRC {X -10.217,Y 74.749,Z -40.000,A 0.015,B -0.000,C -180.000},{X -8.752,Y 74.281,Z -40.000,A 0.015,B 0.000,C -180.000} C_DIS
CIRC {X -6.292,Y 74.711,Z -40.000,A 0.015,B 0.000,C 180.000},{X -5.170,Y 76.941,Z -40.000,A 0.015,B 0.000,C 180.000} C_DIS
LIN {X -5.177,Y 319.913,Z -40.000,A 0.015,B -0.000,C 180.000} C_DIS
CIRC {X -6.306,Y 322.637,Z -40.000,A 0.015,B -0.000,C -180.000},{X -9.030,Y 323.766,Z -40.000,A 0.015,B -0.000,C 180.000} C_DIS
LIN {X -134.620,Y 323.763,Z -40.000,A 0.015,B 0.000,C -180.000} C_DIS
CIRC {X -136.600,Y 322.646,Z -40.000,A 0.015,B 0.000,C 180.000},{X -136.667,Y 320.374,Z -40.000,A 0.015,B -0.000,C 180.000} C_DIS
CIRC {X -133.764,Y 313.950,Z -40.000,A 0.015,B 0.000,C -180.000},{X -131.648,Y 307.226,Z -40.000,A 0.015,B -0.000,C -180.000} C_DIS
CIRC {X -130.761,Y 300.195,Z -40.000,A 0.015,B 0.000,C -180.000},{X -131.560,Y 293.154,Z -40.000,A 0.015,B 0.000,C -180.000} C_DIS
CIRC {X -133.874,Y 284.888,Z -40.000,A 0.015,B 0.000,C 180.000},{X -136.849,Y 276.836,Z -40.000,A 0.015,B 0.000,C -180.000} C_DIS
CIRC {X -141.203,Y 269.358,Z -40.000,A 0.015,B -0.000,C 180.000},{X -147.364,Y 263.283,Z -40.000,A 0.015,B -0.000,C -180.000} C_DIS
CIRC {X -152.265,Y 259.792,Z -40.000,A 0.015,B 0.000,C 180.000},{X -157.345,Y 256.568,Z -40.000,A 0.015,B 0.000,C -180.000} C_DIS
CIRC {X -162.818,Y 254.001,Z -40.000,A 0.015,B 0.000,C -180.000},{X -168.692,Y 252.573,Z -40.000,A 0.015,B 0.000,C -180.000} C_DIS
CIRC {X -171.166,Y 252.209,Z -40.000,A 0.015,B 0.000,C -180.000},{X -173.633,Y 251.804,Z -40.000,A 0.015,B 0.000,C -180.000} C_DIS
CIRC {X -176.116,Y 251.485,Z -40.000,A 0.015,B 0.000,C 180.000},{X -178.617,Y 251.379,Z -40.000,A 0.015,B 0.000,C 180.000} C_DIS
LIN {X -217.564,Y 251.564,Z -40.000,A 0.015,B -0.000,C 180.000} C_DIS
CIRC {X -227.755,Y 253.812,Z -40.000,A 0.015,B 0.000,C 180.000},{X -237.466,Y 257.636,Z -40.000,A 0.015,B -0.000,C 180.000} C_DIS
CIRC {X -246.243,Y 263.372,Z -40.000,A 0.015,B 0.000,C -180.000},{X -253.329,Y 271.101,Z -40.000,A 0.015,B 0.000,C 180.000} C_DIS
CIRC {X -257.799,Y 278.936,Z -40.000,A 0.015,B -0.000,C 180.000},{X -260.643,Y 287.496,Z -40.000,A 0.015,B 0.000,C 180.000} C_DIS
CIRC {X -261.845,Y 295.850,Z -40.000,A 0.015,B -0.000,C 180.000},{X -261.751,Y 304.289,Z -40.000,A 0.015,B 0.000,C -180.000} C_DIS
CIRC {X -260.438,Y 311.563,Z -40.000,A 0.015,B 0.000,C 180.000},{X -257.837,Y 318.482,Z -40.000,A 0.015,B 0.000,C -180.000} C_DIS
CIRC {X -255.304,Y 321.199,Z -40.000,A 0.015,B 0.000,C 180.000},{X -251.678,Y 322.006,Z -40.000,A 0.015,B -0.000,C 180.000} C_DIS
CIRC {X -248.064,Y 322.660,Z -40.000,A 0.015,B 0.000,C -180.000},{X -245.256,Y 325.027,Z -40.000,A 0.015,B 0.000,C 180.000} C_DIS
CIRC {X -243.764,Y 327.007,Z -40.000,A 0.015,B 0.000,C -180.000},{X -242.136,Y 328.877,Z -40.000,A 0.015,B 0.000,C 180.000} C_DIS
CIRC {X -241.803,Y 330.799,Z -40.000,A 0.015,B 0.000,C -180.000},{X -243.434,Y 331.869,Z -40.000,A 0.015,B 0.000,C 180.000} C_DIS
LIN {X -392.601,Y 331.866,Z -40.000,A 0.015,B -0.000,C 180.000} C_DIS
CIRC {X -395.325,Y 330.737,Z -40.000,A 0.015,B -0.000,C -180.000},{X -396.453,Y 328.013,Z -40.000,A 0.015,B -0.000,C 180.000} C_DIS
LIN {X -396.446,Y 62.473,Z -40.000,A 0.015,B -0.000,C -180.000} C_DIS
CIRC {X -395.334,Y 60.699,Z -40.000,A 0.015,B -0.000,C 180.000},{X -393.253,Y 60.928,Z -40.000,A 0.015,B 0.000,C -180.000} C_DIS
CIRC {X -391.494,Y 62.328,Z -40.000,A 0.015,B 0.000,C 180.000},{X -389.743,Y 63.739,Z -40.000,A 0.015,B 0.000,C 180.000} C_DIS
CIRC {X -387.857,Y 64.982,Z -40.000,A 0.015,B 0.000,C -180.000},{X -385.765,Y 65.836,Z -40.000,A 0.015,B -0.000,C -180.000} C_DIS
CIRC {X -380.537,Y 67.321,Z -40.000,A 0.015,B 0.000,C -180.000},{X -375.274,Y 68.673,Z -40.000,A 0.015,B -0.000,C 180.000} C_DIS
CIRC {X -369.856,Y 69.389,Z -40.000,A 0.015,B 0.000,C 180.000},{X -364.409,Y 68.935,Z -40.000,A 0.015,B 0.000,C 180.000} C_DIS
CIRC {X -356.992,Y 66.846,Z -40.000,A 0.015,B 0.000,C -180.000},{X -350.027,Y 63.548,Z -40.000,A 0.015,B 0.000,C -180.000} C_DIS
CIRC {X -343.777,Y 59.021,Z -40.000,A 0.015,B 0.000,C 180.000},{X -338.557,Y 53.336,Z -40.000,A 0.015,B -0.000,C 180.000} C_DIS
LIN {X -317.719,Y 18.116,Z -40.000,A 0.015,B 0.000,C -180.000} C_DIS
CIRC {X -313.907,Y 8.736,Z -40.000,A 0.015,B 0.000,C -180.000},{X -312.770,Y -1.324,Z -40.000,A 0.015,B 0.000,C 180.000} C_DIS
CIRC {X -314.306,Y -11.320,Z -40.000,A 0.015,B -0.000,C -180.000},{X -318.329,Y -20.599,Z -40.000,A 0.015,B 0.000,C 180.000} C_DIS
CIRC {X -318.352,Y -22.817,Z -40.000,A 0.015,B 0.000,C -180.000},{X -316.435,Y -23.933,Z -40.000,A 0.015,B -0.000,C 180.000} C_DIS
LIN {X -77.109,Y -23.933,Z -40.000,A 0.015,B 0.000,C 180.000} C_DIS
CIRC {X -75.172,Y -22.816,Z -40.000,A 0.015,B 0.000,C 180.000},{X -75.167,Y -20.581,Z -40.000,A 0.015,B 0.000,C -180.000} C_DIS
CIRC {X -78.710,Y -12.562,Z -40.000,A 0.015,B 0.000,C 180.000},{X -80.513,Y -3.982,Z -40.000,A 0.015,B 0.000,C 180.000} C_DIS
CIRC {X -80.308,Y 4.805,Z -40.000,A 0.015,B 0.000,C -180.000},{X -77.920,Y 13.264,Z -40.000,A 0.015,B 0.000,C -180.000} C_DIS
LIN {X -57.464,Y 49.891,Z -40.000,A 0.015,B 0.000,C -180.000} C_DIS
CIRC {X -51.419,Y 57.754,Z -40.000,A 0.015,B 0.000,C -180.000},{X -43.540,Y 63.776,Z -40.000,A 0.015,B -0.000,C -180.000} C_DIS
CIRC {X -34.440,Y 67.674,Z -40.000,A 0.015,B 0.000,C 180.000},{X -24.685,Y 69.362,Z -40.000,A 0.015,B 0.000,C 180.000} C_DIS
CIRC {X -19.251,Y 69.225,Z -40.000,A 0.015,B -0.000,C -180.000},{X -13.907,Y 68.223,Z -40.000,A 0.015,B 0.000,C -180.000} C_DIS
CIRC {X -8.776,Y 66.439,Z -40.000,A 0.015,B 0.000,C -180.000},{X -3.942,Y 63.961,Z -40.000,A 0.015,B 0.000,C -180.000} C_DIS
CIRC {X -2.952,Y 63.285,Z -40.000,A 0.015,B 0.000,C 180.000},{X -2.043,Y 62.503,Z -40.000,A 0.015,B 0.000,C 180.000} C_DIS
CIRC {X -1.161,Y 61.692,Z -40.000,A 0.015,B 0.000,C -180.000},{X -0.245,Y 60.920,Z -40.000,A 0.015,B 0.000,C -180.000} C_DIS
CIRC {X 1.827,Y 60.680,Z -40.000,A 0.015,B 0.000,C -180.000},{X 2.939,Y 62.445,Z -40.000,A 0.015,B 0.000,C -180.000} C_DIS
LIN {X 2.932,Y 328.022,Z -40.000,A 0.015,B 0.000,C 180.000} C_DIS
CIRC {X 1.803,Y 330.747,Z -40.000,A 0.015,B 0.000,C -180.000},{X -0.921,Y 331.875,Z -40.000,A 0.015,B 0.000,C -180.000} C_DIS
LIN {X -150.043,Y 331.872,Z -40.000,A 0.015,B -0.000,C -180.000} C_DIS
CIRC {X -151.710,Y 330.765,Z -40.000,A 0.015,B -0.000,C 180.000},{X -151.338,Y 328.799,Z -40.000,A 0.015,B 0.000,C 180.000} C_DIS
CIRC {X -145.990,Y 322.136,Z -40.000,A 0.015,B 0.000,C 180.000},{X -142.014,Y 314.574,Z -40.000,A 0.015,B 0.000,C 180.000} C_DIS
CIRC {X -139.655,Y 306.351,Z -40.000,A 0.015,B 0.000,C 180.000},{X -139.127,Y 297.812,Z -40.000,A 0.015,B 0.000,C -180.000} C_DIS
CIRC {X -141.281,Y 286.319,Z -40.000,A 0.015,B -0.000,C 180.000},{X -146.494,Y 275.853,Z -40.000,A 0.015,B -0.000,C -180.000} C_DIS
CIRC {X -154.618,Y 267.380,Z -40.000,A 0.015,B 0.000,C 180.000},{X -165.038,Y 261.974,Z -40.000,A 0.015,B 0.000,C -180.000} C_DIS
CIRC {X -168.359,Y 260.993,Z -40.000,A 0.015,B 0.000,C 180.000},{X -171.729,Y 260.196,Z -40.000,A 0.015,B 0.000,C 180.000} C_DIS
CIRC {X -175.155,Y 259.665,Z -40.000,A 0.015,B 0.000,C -180.000},{X -178.617,Y 259.488,Z -40.000,A 0.015,B 0.000,C 180.000} C_DIS
LIN {X -216.447,Y 259.595,Z -40.000,A 0.015,B 0.000,C -180.000} C_DIS
CIRC {X -225.037,Y 261.452,Z -40.000,A 0.015,B -0.000,C 180.000},{X -233.256,Y 264.566,Z -40.000,A 0.015,B 0.000,C 180.000} C_DIS
CIRC {X -240.715,Y 269.305,Z -40.000,A 0.015,B 0.000,C -180.000},{X -246.716,Y 275.794,Z -40.000,A 0.015,B 0.000,C 180.000} C_DIS
CIRC {X -250.389,Y 282.232,Z -40.000,A 0.015,B 0.000,C -180.000},{X -252.729,Y 289.264,Z -40.000,A 0.015,B -0.000,C 180.000} C_DIS
CIRC {X -253.814,Y 296.024,Z -40.000,A 0.015,B 0.000,C -180.000},{X -254.072,Y 302.866,Z -40.000,A 0.015,B 0.000,C 180.000} C_DIS
CIRC {X -253.093,Y 309.679,Z -40.000,A 0.015,B 0.000,C 180.000},{X -250.523,Y 316.064,Z -40.000,A 0.015,B 0.000,C -180.000} C_DIS
CIRC {X -248.651,Y 319.412,Z -40.000,A 0.015,B 0.000,C 180.000},{X -246.730,Y 322.732,Z -40.000,A 0.015,B 0.000,C -180.000} C_DIS
CIRC {X -246.015,Y 323.894,Z -40.000,A 0.015,B 0.000,C -180.000},{X -245.256,Y 325.027,Z -40.000,A 0.015,B 0.000,C 180.000} C_DIS
LIN {X -245.084,Y 325.631,Z -39.830,A 0.015,B 0.000,C 180.000} C_DIS
LIN {X -245.155,Y 326.088,Z -39.365,A 0.015,B 0.000,C -180.000} C_DIS
LIN {X -245.222,Y 326.244,Z -38.730,A 0.015,B 0.000,C -180.000} C_DIS
$VEL.CP = 1.00000
LIN {X -245.222,Y 326.244,Z 11.000,A 0.015,B 0.000,C 180.000} C_DIS
$VEL.CP = 1.00000
LIN {X -398.499,Y 339.199,Z 11.000,A 0.015,B 0.000,C -180.000} C_DIS
$VEL.CP = 0.10000
LIN {X -398.499,Y 339.199,Z -18.231,A 0.015,B -0.000,C -180.000} C_DIS
LIN {X -398.507,Y 339.199,Z -18.374,A 0.015,B 0.000,C -180.000} C_DIS
LIN {X -398.772,Y 339.192,Z -19.019,A 0.015,B -0.000,C -180.000} C_DIS
LIN {X -399.336,Y 339.133,Z -19.426,A 0.015,B 0.000,C -180.000} C_DIS
LIN {X -399.692,Y 339.076,Z -19.499,A 0.015,B -0.000,C -180.000} C_DIS
LIN {X -399.716,Y 339.073,Z -19.500,A 0.015,B 0.000,C -180.000} C_DIS
LIN {X -400.552,Y 338.848,Z -19.530,A 0.015,B 0.000,C -180.000} C_DIS
LIN {X -400.596,Y 338.832,Z -19.532,A 0.015,B 0.000,C -180.000} C_DIS
LIN {X -401.281,Y 338.494,Z -19.559,A 0.015,B -0.000,C -180.000} C_DIS
LIN {X -401.404,Y 338.418,Z -19.564,A 0.015,B 0.000,C -180.000} C_DIS
LIN {X -402.842,Y 337.053,Z -19.633,A 0.015,B -0.000,C 180.000} C_DIS
LIN {X -402.866,Y 337.018,Z -19.635,A 0.015,B 0.000,C -180.000} C_DIS
LIN {X -403.753,Y 334.430,Z -19.732,A 0.015,B 0.000,C 180.000} C_DIS
LIN {X -403.779,Y 333.946,Z -19.749,A 0.015,B -0.000,C -180.000} C_DIS
LIN {X -403.787,Y 333.653,Z -19.759,A 0.015,B -0.000,C -180.000} C_DIS
LIN {X -403.787,Y 333.050,Z -19.780,A 0.015,B 0.000,C -180.000} C_DIS
LIN {X -401.252,Y 328.076,Z -19.982,A 0.015,B -0.000,C -180.000} C_DIS
LIN {X -395.738,Y 327.203,Z -20.185,A 0.015,B -0.000,C -180.000} C_DIS
LIN {X -391.790,Y 331.150,Z -20.387,A 0.015,B -0.000,C -180.000} C_DIS
LIN {X -392.664,Y 336.664,Z -20.589,A 0.015,B 0.000,C 180.000} C_DIS
LIN {X -397.638,Y 339.199,Z -20.792,A 0.015,B 0.000,C -180.000} C_DIS
LIN {X -398.507,Y 339.199,Z -20.822,A 0.015,B -0.000,C -180.000} C_DIS
LIN {X -399.336,Y 339.133,Z -20.851,A 0.015,B -0.000,C -180.000} C_DIS
LIN {X -399.692,Y 339.076,Z -20.864,A 0.015,B 0.000,C 180.000} C_DIS
LIN {X -400.552,Y 338.848,Z -20.895,A 0.015,B 0.000,C -180.000} C_DIS
LIN {X -400.596,Y 338.832,Z -20.896,A 0.015,B -0.000,C -180.000} C_DIS
LIN {X -401.281,Y 338.494,Z -20.923,A 0.015,B -0.000,C -180.000} C_DIS
LIN {X -401.404,Y 338.418,Z -20.928,A 0.015,B -0.000,C -180.000} C_DIS
LIN {X -402.842,Y 337.053,Z -20.998,A 0.015,B -0.000,C -180.000} C_DIS
LIN {X -402.866,Y 337.018,Z -20.999,A 0.015,B -0.000,C -180.000} C_DIS
LIN {X -403.753,Y 334.430,Z -21.096,A 0.015,B -0.000,C -180.000} C_DIS
LIN {X -403.779,Y 333.946,Z -21.113,A 0.015,B 0.000,C -180.000} C_DIS
LIN {X -403.787,Y 333.653,Z -21.123,A 0.015,B -0.000,C 180.000} C_DIS
LIN {X -403.787,Y 333.050,Z -21.144,A 0.015,B -0.000,C -180.000} C_DIS
LIN {X -401.252,Y 328.076,Z -21.347,A 0.015,B 0.000,C -180.000} C_DIS
LIN {X -395.738,Y 327.203,Z -21.549,A 0.015,B 0.000,C 180.000} C_DIS
LIN {X -391.790,Y 331.150,Z -21.752,A 0.015,B -0.000,C 180.000} C_DIS
LIN {X -392.664,Y 336.664,Z -21.954,A 0.015,B -0.000,C -180.000} C_DIS
LIN {X -397.638,Y 339.199,Z -22.156,A 0.015,B -0.000,C -180.000} C_DIS
LIN {X -398.507,Y 339.199,Z -22.187,A 0.015,B -0.000,C -180.000} C_DIS
LIN {X -399.336,Y 339.133,Z -22.216,A 0.015,B 0.000,C 180.000} C_DIS
LIN {X -399.692,Y 339.076,Z -22.228,A 0.015,B -0.000,C -180.000} C_DIS
LIN {X -400.552,Y 338.848,Z -22.259,A 0.015,B 0.000,C 180.000} C_DIS
LIN {X -400.596,Y 338.832,Z -22.261,A 0.015,B 0.000,C -180.000} C_DIS
LIN {X -401.281,Y 338.494,Z -22.288,A 0.015,B 0.000,C -180.000} C_DIS
LIN {X -401.404,Y 338.418,Z -22.293,A 0.015,B 0.000,C -180.000} C_DIS
LIN {X -402.842,Y 337.053,Z -22.362,A 0.015,B 0.000,C -180.000} C_DIS
LIN {X -402.866,Y 337.018,Z -22.364,A 0.015,B 0.000,C -180.000} C_DIS
LIN {X -403.753,Y 334.430,Z -22.461,A 0.015,B 0.000,C -180.000} C_DIS
LIN {X -403.779,Y 333.946,Z -22.478,A 0.015,B -0.000,C -180.000} C_DIS
LIN {X -403.787,Y 333.653,Z -22.488,A 0.015,B -0.000,C -180.000} C_DIS
LIN {X -403.787,Y 333.050,Z -22.509,A 0.015,B 0.000,C -180.000} C_DIS
LIN {X -401.252,Y 328.076,Z -22.711,A 0.015,B -0.000,C 180.000} C_DIS
LIN {X -395.738,Y 327.203,Z -22.914,A 0.015,B 0.000,C 180.000} C_DIS
LIN {X -391.790,Y 331.150,Z -23.116,A 0.015,B -0.000,C 180.000} C_DIS
LIN {X -392.664,Y 336.664,Z -23.318,A 0.015,B -0.000,C -180.000} C_DIS
LIN {X -397.638,Y 339.199,Z -23.521,A 0.015,B 0.000,C 180.000} C_DIS
LIN {X -398.507,Y 339.199,Z -23.551,A 0.015,B 0.000,C 180.000} C_DIS
LIN {X -399.336,Y 339.133,Z -23.580,A 0.015,B -0.000,C 180.000} C_DIS
LIN {X -399.692,Y 339.076,Z -23.593,A 0.015,B -0.000,C 180.000} C_DIS
LIN {X -400.552,Y 338.848,Z -23.624,A 0.015,B -0.000,C -180.000} C_DIS
LIN {X -400.596,Y 338.832,Z -23.626,A 0.015,B -0.000,C -180.000} C_DIS
LIN {X -401.281,Y 338.494,Z -23.652,A 0.015,B -0.000,C -180.000} C_DIS
LIN {X -401.404,Y 338.418,Z -23.657,A 0.015,B -0.000,C 180.000} C_DIS
LIN {X -402.842,Y 337.053,Z -23.727,A 0.015,B -0.000,C 180.000} C_DIS
LIN {X -402.866,Y 337.018,Z -23.728,A 0.015,B -0.000,C -180.000} C_DIS
LIN {X -403.753,Y 334.430,Z -23.825,A 0.015,B -0.000,C -180.000} C_DIS
LIN {X -403.779,Y 333.946,Z -23.842,A 0.015,B 0.000,C -180.000} C_DIS
LIN {X -403.787,Y 333.653,Z -23.852,A 0.015,B -0.000,C 180.000} C_DIS
LIN {X -403.787,Y 333.050,Z -23.873,A 0.015,B 0.000,C -180.000} C_DIS
LIN {X -401.252,Y 328.076,Z -24.076,A 0.015,B 0.000,C -180.000} C_DIS
LIN {X -395.738,Y 327.203,Z -24.278,A 0.015,B -0.000,C -180.000} C_DIS
LIN {X -391.790,Y 331.150,Z -24.481,A 0.015,B 0.000,C -180.000} C_DIS
LIN {X -392.664,Y 336.664,Z -24.683,A 0.015,B 0.000,C -180.000} C_DIS
LIN {X -397.638,Y 339.199,Z -24.885,A 0.015,B 0.000,C 180.000} C_DIS
LIN {X -398.507,Y 339.199,Z -24.916,A 0.015,B 0.000,C -180.000} C_DIS
LIN {X -399.336,Y 339.133,Z -24.945,A 0.015,B 0.000,C -180.000} C_DIS
LIN {X -399.692,Y 339.076,Z -24.957,A 0.015,B 0.000,C 180.000} C_DIS
LIN {X -400.552,Y 338.848,Z -24.988,A 0.015,B 0.000,C 180.000} C_DIS
LIN {X -400.596,Y 338.832,Z -24.990,A 0.015,B 0.000,C -180.000} C_DIS
LIN {X -401.281,Y 338.494,Z -25.017,A 0.015,B 0.000,C -180.000} C_DIS
LIN {X -401.404,Y 338.418,Z -25.022,A 0.015,B -0.000,C -180.000} C_DIS
LIN {X -402.842,Y 337.053,Z -25.092,A 0.015,B 0.000,C -180.000} C_DIS
LIN {X -402.866,Y 337.018,Z -25.093,A 0.015,B 0.000,C 180.000} C_DIS
LIN {X -403.753,Y 334.430,Z -25.190,A 0.015,B 0.000,C -180.000} C_DIS
LIN {X -403.779,Y 333.946,Z -25.207,A 0.015,B 0.000,C 180.000} C_DIS
LIN {X -403.787,Y 333.653,Z -25.217,A 0.015,B -0.000,C 180.000} C_DIS
LIN {X -403.787,Y 333.050,Z -25.238,A 0.015,B -0.000,C -180.000} C_DIS
LIN {X -401.252,Y 328.076,Z -25.440,A 0.015,B -0.000,C -180.000} C_DIS
LIN {X -395.738,Y 327.203,Z -25.643,A 0.015,B 0.000,C 180.000} C_DIS
LIN {X -391.790,Y 331.150,Z -25.845,A 0.015,B 0.000,C -180.000} C_DIS
LIN {X -392.664,Y 336.664,Z -26.047,A 0.015,B 0.000,C 180.000} C_DIS
LIN {X -397.638,Y 339.199,Z -26.250,A 0.015,B -0.000,C -180.000} C_DIS
LIN {X -398.507,Y 339.199,Z -26.280,A 0.015,B 0.000,C 180.000} C_DIS
LIN {X -399.336,Y 339.133,Z -26.309,A 0.015,B -0.000,C 180.000} C_DIS
LIN {X -399.692,Y 339.076,Z -26.322,A 0.015,B -0.000,C 180.000} C_DIS
LIN {X -400.552,Y 338.848,Z -26.353,A 0.015,B 0.000,C 180.000} C_DIS
LIN {X -400.596,Y 338.832,Z -26.355,A 0.015,B -0.000,C 180.000} C_DIS
LIN {X -401.281,Y 338.494,Z -26.381,A 0.015,B 0.000,C -180.000} C_DIS
LIN {X -401.404,Y 338.418,Z -26.386,A 0.015,B 0.000,C 180.000} C_DIS
LIN {X -402.842,Y 337.053,Z -26.456,A 0.015,B -0.000,C -180.000} C_DIS
LIN {X -402.866,Y 337.018,Z -26.458,A 0.015,B -0.000,C -180.000} C_DIS
LIN {X -403.753,Y 334.430,Z -26.554,A 0.015,B -0.000,C 180.000} C_DIS
LIN {X -403.779,Y 333.946,Z -26.571,A 0.015,B -0.000,C -180.000} C_DIS
LIN {X -403.787,Y 333.653,Z -26.582,A 0.015,B -0.000,C 180.000} C_DIS
LIN {X -403.787,Y 333.050,Z -26.603,A 0.015,B -0.000,C -180.000} C_DIS
LIN {X -401.252,Y 328.076,Z -26.805,A 0.015,B 0.000,C 180.000} C_DIS
LIN {X -395.738,Y 327.203,Z -27.007,A 0.015,B -0.000,C -180.000} C_DIS
LIN {X -391.790,Y 331.150,Z -27.210,A 0.015,B -0.000,C 180.000} C_DIS
LIN {X -392.664,Y 336.664,Z -27.412,A 0.015,B -0.000,C 180.000} C_DIS
LIN {X -397.638,Y 339.199,Z -27.614,A 0.015,B 0.000,C -180.000} C_DIS
LIN {X -398.507,Y 339.199,Z -27.645,A 0.015,B 0.000,C -180.000} C_DIS
LIN {X -399.336,Y 339.133,Z -27.674,A 0.015,B 0.000,C -180.000} C_DIS
LIN {X -399.692,Y 339.076,Z -27.686,A 0.015,B -0.000,C -180.000} C_DIS
LIN {X -400.552,Y 338.848,Z -27.718,A 0.015,B 0.000,C 180.000} C_DIS
LIN {X -400.596,Y 338.832,Z -27.719,A 0.015,B -0.000,C -180.000} C_DIS
LIN {X -401.281,Y 338.494,Z -27.746,A 0.015,B -0.000,C -180.000} C_DIS
LIN {X -401.404,Y 338.418,Z -27.751,A 0.015,B 0.000,C 180.000} C_DIS
LIN {X -402.842,Y 337.053,Z -27.821,A 0.015,B 0.000,C -180.000} C_DIS
LIN {X -402.866,Y 337.018,Z -27.822,A 0.015,B -0.000,C -180.000} C_DIS
LIN {X -403.753,Y 334.430,Z -27.919,A 0.015,B -0.000,C -180.000} C_DIS
LIN {X -403.779,Y 333.946,Z -27.936,A 0.015,B 0.000,C -180.000} C_DIS
LIN {X -403.787,Y 333.653,Z -27.946,A 0.015,B -0.000,C -180.000} C_DIS
LIN {X -403.787,Y 333.050,Z -27.967,A 0.015,B 0.000,C -180.000} C_DIS
LIN {X -401.252,Y 328.076,Z -28.169,A 0.015,B 0.000,C -180.000} C_DIS
LIN {X -395.738,Y 327.203,Z -28.372,A 0.015,B 0.000,C -180.000} C_DIS
LIN {X -391.790,Y 331.150,Z -28.574,A 0.015,B 0.000,C -180.000} C_DIS
LIN {X -392.664,Y 336.664,Z -28.777,A 0.015,B -0.000,C -180.000} C_DIS
LIN {X -397.638,Y 339.199,Z -28.979,A 0.015,B -0.000,C -180.000} C_DIS
LIN {X -398.507,Y 339.199,Z -29.009,A 0.015,B -0.000,C -180.000} C_DIS
LIN {X -399.336,Y 339.133,Z -29.038,A 0.015,B 0.000,C -180.000} C_DIS
LIN {X -399.692,Y 339.076,Z -29.051,A 0.015,B 0.000,C -180.000} C_DIS
LIN {X -400.552,Y 338.848,Z -29.082,A 0.015,B 0.000,C -180.000} C_DIS
LIN {X -400.596,Y 338.832,Z -29.084,A 0.015,B 0.000,C -180.000} C_DIS
LIN {X -401.281,Y 338.494,Z -29.110,A 0.015,B 0.000,C 180.000} C_DIS
LIN {X -401.404,Y 338.418,Z -29.115,A 0.015,B 0.000,C 180.000} C_DIS
LIN {X -402.842,Y 337.053,Z -29.185,A 0.015,B 0.000,C -180.000} C_DIS
LIN {X -402.866,Y 337.018,Z -29.187,A 0.015,B 0.000,C -180.000} C_DIS
LIN {X -403.753,Y 334.430,Z -29.283,A 0.015,B 0.000,C 180.000} C_DIS
LIN {X -403.779,Y 333.946,Z -29.300,A 0.015,B -0.000,C -180.000} C_DIS
LIN {X -403.787,Y 333.653,Z -29.311,A 0.015,B 0.000,C -180.000} C_DIS
LIN {X -403.787,Y 333.050,Z -29.332,A 0.015,B 0.000,C -180.000} C_DIS
LIN {X -401.252,Y 328.076,Z -29.534,A 0.015,B 0.000,C -180.000} C_DIS
LIN {X -395.738,Y 327.203,Z -29.736,A 0.015,B 0.000,C -180.000} C_DIS
LIN {X -391.790,Y 331.150,Z -29.939,A 0.015,B -0.000,C -180.000} C_DIS
LIN {X -392.664,Y 336.664,Z -30.141,A 0.015,B 0.000,C -180.000} C_DIS
LIN {X -397.638,Y 339.199,Z -30.343,A 0.015,B -0.000,C -180.000} C_DIS
LIN {X -398.507,Y 339.199,Z -30.374,A 0.015,B -0.000,C -180.000} C_DIS
LIN {X -399.336,Y 339.133,Z -30.403,A 0.015,B 0.000,C -180.000} C_DIS
LIN {X -399.692,Y 339.076,Z -30.415,A 0.015,B -0.000,C -180.000} C_DIS
LIN {X -400.552,Y 338.848,Z -30.447,A 0.015,B 0.000,C 180.000} C_DIS
LIN {X -400.596,Y 338.832,Z -30.448,A 0.015,B -0.000,C 180.000} C_DIS
LIN {X -401.281,Y 338.494,Z -30.475,A 0.015,B -0.000,C -180.000} C_DIS
LIN {X -401.404,Y 338.418,Z -30.480,A 0.015,B 0.000,C -180.000} C_DIS
LIN {X -402.842,Y 337.053,Z -30.550,A 0.015,B -0.000,C -180.000} C_DIS
LIN {X -402.866,Y 337.018,Z -30.551,A 0.015,B -0.000,C -180.000} C_DIS
LIN {X -403.753,Y 334.430,Z -30.648,A 0.015,B 0.000,C -180.000} C_DIS
LIN {X -403.779,Y 333.946,Z -30.665,A 0.015,B 0.000,C 180.000} C_DIS
LIN {X -403.787,Y 333.653,Z -30.675,A 0.015,B 0.000,C -180.000} C_DIS
LIN {X -403.787,Y 333.050,Z -30.696,A 0.015,B 0.000,C -180.000} C_DIS
LIN {X -401.252,Y 328.076,Z -30.899,A 0.015,B 0.000,C 180.000} C_DIS
LIN {X -395.738,Y 327.203,Z -31.101,A 0.015,B -0.000,C 180.000} C_DIS
LIN {X -391.790,Y 331.150,Z -31.303,A 0.015,B -0.000,C -180.000} C_DIS
LIN {X -392.664,Y 336.664,Z -31.506,A 0.015,B 0.000,C 180.000} C_DIS
LIN {X -397.638,Y 339.199,Z -31.708,A 0.015,B -0.000,C -180.000} C_DIS
LIN {X -398.507,Y 339.199,Z -31.738,A 0.015,B -0.000,C 180.000} C_DIS
LIN {X -399.336,Y 339.133,Z -31.767,A 0.015,B 0.000,C 180.000} C_DIS
LIN {X -399.692,Y 339.076,Z -31.780,A 0.015,B 0.000,C -180.000} C_DIS
LIN {X -400.552,Y 338.848,Z -31.811,A 0.015,B -0.000,C -180.000} C_DIS
LIN {X -400.596,Y 338.832,Z -31.813,A 0.015,B -0.000,C -180.000} C_DIS
LIN {X -401.281,Y 338.494,Z -31.839,A 0.015,B 0.000,C 180.000} C_DIS
LIN {X -401.404,Y 338.418,Z -31.845,A 0.015,B -0.000,C -180.000} C_DIS
LIN {X -402.842,Y 337.053,Z -31.914,A 0.015,B 0.000,C -180.000} C_DIS
LIN {X -402.866,Y 337.018,Z -31.916,A 0.015,B -0.000,C -180.000} C_DIS
LIN {X -403.753,Y 334.430,Z -32.013,A 0.015,B -0.000,C -180.000} C_DIS
LIN {X -403.779,Y 333.946,Z -32.029,A 0.015,B -0.000,C -180.000} C_DIS
LIN {X -403.787,Y 333.653,Z -32.040,A 0.015,B -0.000,C -180.000} C_DIS
LIN {X -403.787,Y 333.050,Z -32.061,A 0.015,B 0.000,C 180.000} C_DIS
LIN {X -401.252,Y 328.076,Z -32.263,A 0.015,B 0.000,C 180.000} C_DIS
LIN {X -395.738,Y 327.203,Z -32.465,A 0.015,B -0.000,C -180.000} C_DIS
LIN {X -391.790,Y 331.150,Z -32.668,A 0.015,B -0.000,C 180.000} C_DIS
LIN {X -392.664,Y 336.664,Z -32.870,A 0.015,B 0.000,C -180.000} C_DIS
LIN {X -397.638,Y 339.199,Z -33.073,A 0.015,B 0.000,C -180.000} C_DIS
LIN {X -398.507,Y 339.199,Z -33.103,A 0.015,B -0.000,C 180.000} C_DIS
LIN {X -399.336,Y 339.133,Z -33.132,A 0.015,B 0.000,C -180.000} C_DIS
LIN {X -399.692,Y 339.076,Z -33.145,A 0.015,B 0.000,C 180.000} C_DIS
LIN {X -400.552,Y 338.848,Z -33.176,A 0.015,B 0.000,C 180.000} C_DIS
LIN {X -400.596,Y 338.832,Z -33.177,A 0.015,B -0.000,C -180.000} C_DIS
LIN {X -401.281,Y 338.494,Z -33.204,A 0.015,B -0.000,C -180.000} C_DIS
LIN {X -401.404,Y 338.418,Z -33.209,A 0.015,B 0.000,C -180.000} C_DIS
LIN {X -402.842,Y 337.053,Z -33.279,A 0.015,B 0.000,C 180.000} C_DIS
LIN {X -402.866,Y 337.018,Z -33.280,A 0.015,B 0.000,C -180.000} C_DIS
LIN {X -403.753,Y 334.430,Z -33.377,A 0.015,B -0.000,C -180.000} C_DIS
LIN {X -403.779,Y 333.946,Z -33.394,A 0.015,B 0.000,C -180.000} C_DIS
LIN {X -403.787,Y 333.653,Z -33.404,A 0.015,B -0.000,C -180.000} C_DIS
LIN {X -403.787,Y 333.050,Z -33.425,A 0.015,B 0.000,C 180.000} C_DIS
LIN {X -401.252,Y 328.076,Z -33.628,A 0.015,B 0.000,C -180.000} C_DIS
LIN {X -395.738,Y 327.203,Z -33.830,A 0.015,B -0.000,C -180.000} C_DIS
LIN {X -391.790,Y 331.150,Z -34.032,A 0.015,B -0.000,C -180.000} C_DIS
LIN {X -392.664,Y 336.664,Z -34.235,A 0.015,B -0.000,C 180.000} C_DIS
LIN {X -397.638,Y 339.199,Z -34.437,A 0.015,B 0.000,C -180.000} C_DIS
LIN {X -398.507,Y 339.199,Z -34.467,A 0.015,B -0.000,C -180.000} C_DIS
LIN {X -399.336,Y 339.133,Z -34.496,A 0.015,B 0.000,C 180.000} C_DIS
LIN {X -399.692,Y 339.076,Z -34.509,A 0.015,B 0.000,C -180.000} C_DIS
LIN {X -400.552,Y 338.848,Z -34.540,A 0.015,B 0.000,C 180.000} C_DIS
LIN {X -400.596,Y 338.832,Z -34.542,A 0.015,B 0.000,C 180.000} C_DIS
LIN {X -401.281,Y 338.494,Z -34.569,A 0.015,B 0.000,C -180.000} C_DIS
LIN {X -401.404,Y 338.418,Z -34.574,A 0.015,B -0.000,C -180.000} C_DIS
LIN {X -402.842,Y 337.053,Z -34.643,A 0.015,B 0.000,C -180.000} C_DIS
LIN {X -402.866,Y 337.018,Z -34.645,A 0.015,B -0.000,C -180.000} C_DIS
LIN {X -403.753,Y 334.430,Z -34.742,A 0.015,B 0.000,C -180.000} C_DIS
LIN {X -403.779,Y 333.946,Z -34.759,A 0.015,B -0.000,C -180.000} C_DIS
LIN {X -403.787,Y 333.653,Z -34.769,A 0.015,B -0.000,C -180.000} C_DIS
LIN {X -403.787,Y 333.050,Z -34.790,A 0.015,B 0.000,C -180.000} C_DIS
LIN {X -401.252,Y 328.076,Z -34.992,A 0.015,B 0.000,C -180.000} C_DIS
LIN {X -395.738,Y 327.203,Z -35.195,A 0.015,B -0.000,C 180.000} C_DIS
LIN {X -391.790,Y 331.150,Z -35.397,A 0.015,B 0.000,C 180.000} C_DIS
LIN {X -392.664,Y 336.664,Z -35.599,A 0.015,B 0.000,C 180.000} C_DIS
LIN {X -397.638,Y 339.199,Z -35.802,A 0.015,B -0.000,C 180.000} C_DIS
LIN {X -398.507,Y 339.199,Z -35.832,A 0.015,B 0.000,C -180.000} C_DIS
LIN {X -399.336,Y 339.133,Z -35.861,A 0.015,B -0.000,C -180.000} C_DIS
LIN {X -399.692,Y 339.076,Z -35.874,A 0.015,B -0.000,C -180.000} C_DIS
LIN {X -400.552,Y 338.848,Z -35.905,A 0.015,B -0.000,C -180.000} C_DIS
LIN {X -400.596,Y 338.832,Z -35.906,A 0.015,B 0.000,C -180.000} C_DIS
LIN {X -401.281,Y 338.494,Z -35.933,A 0.015,B 0.000,C -180.000} C_DIS
LIN {X -401.404,Y 338.418,Z -35.938,A 0.015,B 0.000,C -180.000} C_DIS
LIN {X -402.842,Y 337.053,Z -36.008,A 0.015,B 0.000,C -180.000} C_DIS
LIN {X -402.866,Y 337.018,Z -36.009,A 0.015,B -0.000,C -180.000} C_DIS
LIN {X -403.753,Y 334.430,Z -36.106,A 0.015,B -0.000,C -180.000} C_DIS
LIN {X -403.779,Y 333.946,Z -36.123,A 0.015,B -0.000,C -180.000} C_DIS
LIN {X -403.787,Y 333.653,Z -36.133,A 0.015,B -0.000,C -180.000} C_DIS
LIN {X -403.787,Y 333.050,Z -36.154,A 0.015,B -0.000,C -180.000} C_DIS
LIN {X -401.252,Y 328.076,Z -36.357,A 0.015,B 0.000,C -180.000} C_DIS
LIN {X -395.738,Y 327.203,Z -36.559,A 0.015,B -0.000,C 180.000} C_DIS
LIN {X -391.790,Y 331.150,Z -36.761,A 0.015,B 0.000,C -180.000} C_DIS
LIN {X -392.664,Y 336.664,Z -36.964,A 0.015,B -0.000,C 180.000} C_DIS
LIN {X -397.638,Y 339.199,Z -37.166,A 0.015,B 0.000,C -180.000} C_DIS
LIN {X -398.507,Y 339.199,Z -37.196,A 0.015,B -0.000,C -180.000} C_DIS
LIN {X -399.336,Y 339.133,Z -37.226,A 0.015,B 0.000,C -180.000} C_DIS
LIN {X -399.692,Y 339.076,Z -37.238,A 0.015,B 0.000,C -180.000} C_DIS
LIN {X -400.552,Y 338.848,Z -37.269,A 0.015,B -0.000,C 180.000} C_DIS
LIN {X -400.596,Y 338.832,Z -37.271,A 0.015,B 0.000,C -180.000} C_DIS
LIN {X -401.281,Y 338.494,Z -37.298,A 0.015,B -0.000,C 180.000} C_DIS
LIN {X -401.404,Y 338.418,Z -37.303,A 0.015,B -0.000,C -180.000} C_DIS
LIN {X -402.842,Y 337.053,Z -37.372,A 0.015,B -0.000,C -180.000} C_DIS
LIN {X -402.866,Y 337.018,Z -37.374,A 0.015,B -0.000,C -180.000} C_DIS
LIN {X -403.753,Y 334.430,Z -37.471,A 0.015,B -0.000,C 180.000} C_DIS
LIN {X -403.779,Y 333.946,Z -37.488,A 0.015,B 0.000,C -180.000} C_DIS
LIN {X -403.787,Y 333.653,Z -37.498,A 0.015,B 0.000,C 180.000} C_DIS
LIN {X -403.787,Y 333.050,Z -37.519,A 0.015,B -0.000,C 180.000} C_DIS
LIN {X -401.252,Y 328.076,Z -37.721,A 0.015,B 0.000,C -180.000} C_DIS
LIN {X -395.738,Y 327.203,Z -37.924,A 0.015,B 0.000,C 180.000} C_DIS
LIN {X -391.790,Y 331.150,Z -38.126,A 0.015,B 0.000,C -180.000} C_DIS
LIN {X -392.664,Y 336.664,Z -38.328,A 0.015,B 0.000,C -180.000} C_DIS
LIN {X -397.638,Y 339.199,Z -38.531,A 0.015,B 0.000,C -180.000} C_DIS
LIN {X -398.507,Y 339.199,Z -38.561,A 0.015,B 0.000,C -180.000} C_DIS
LIN {X -399.336,Y 339.133,Z -38.590,A 0.015,B -0.000,C -180.000} C_DIS
LIN {X -399.692,Y 339.076,Z -38.603,A 0.015,B -0.000,C 180.000} C_DIS
LIN {X -400.552,Y 338.848,Z -38.634,A 0.015,B -0.000,C 180.000} C_DIS
LIN {X -400.596,Y 338.832,Z -38.635,A 0.015,B -0.000,C -180.000} C_DIS
LIN {X -401.281,Y 338.494,Z -38.662,A 0.015,B 0.000,C -180.000} C_DIS
LIN {X -401.404,Y 338.418,Z -38.667,A 0.015,B 0.000,C -180.000} C_DIS
LIN {X -402.842,Y 337.053,Z -38.737,A 0.015,B -0.000,C -180.000} C_DIS
LIN {X -402.866,Y 337.018,Z -38.738,A 0.015,B 0.000,C -180.000} C_DIS
LIN {X -403.753,Y 334.430,Z -38.835,A 0.015,B 0.000,C -180.000} C_DIS
LIN {X -403.779,Y 333.946,Z -38.852,A 0.015,B 0.000,C -180.000} C_DIS
LIN {X -403.787,Y 333.653,Z -38.862,A 0.015,B -0.000,C -180.000} C_DIS
LIN {X -403.787,Y 333.050,Z -38.883,A 0.015,B 0.000,C -180.000} C_DIS
LIN {X -401.252,Y 328.076,Z -39.086,A 0.015,B 0.000,C 180.000} C_DIS
LIN {X -395.738,Y 327.203,Z -39.288,A 0.015,B -0.000,C -180.000} C_DIS
LIN {X -391.790,Y 331.150,Z -39.491,A 0.015,B -0.000,C -180.000} C_DIS
LIN {X -392.664,Y 336.664,Z -39.693,A 0.015,B 0.000,C 180.000} C_DIS
LIN {X -397.638,Y 339.199,Z -39.895,A 0.015,B -0.000,C -180.000} C_DIS
LIN {X -398.507,Y 339.199,Z -39.926,A 0.015,B 0.000,C -180.000} C_DIS
LIN {X -399.336,Y 339.133,Z -39.955,A 0.015,B 0.000,C -180.000} C_DIS
LIN {X -399.692,Y 339.076,Z -39.967,A 0.015,B 0.000,C -180.000} C_DIS
LIN {X -400.552,Y 338.848,Z -39.998,A 0.015,B 0.000,C -180.000} C_DIS
LIN {X -400.596,Y 338.832,Z -40.000,A 0.015,B 0.000,C -180.000} C_DIS
LIN {X -400.134,Y 339.006,Z -40.000,A 0.015,B -0.000,C -180.000} C_DIS
LIN {X -398.924,Y 339.199,Z -40.000,A 0.015,B 0.000,C -180.000} C_DIS
LIN {X -213.352,Y 339.203,Z -40.000,A 0.015,B 0.000,C 180.000} C_DIS
LIN {X -213.546,Y 339.161,Z -40.000,A 0.015,B -0.000,C 180.000} C_DIS
LIN {X -214.634,Y 338.886,Z -40.000,A 0.015,B -0.000,C 180.000} C_DIS
LIN {X -215.282,Y 338.650,Z -40.000,A 0.015,B -0.000,C 180.000} C_DIS
LIN {X -225.803,Y 333.552,Z -40.000,A 0.015,B 0.000,C -180.000} C_DIS
LIN {X -226.114,Y 333.381,Z -40.000,A 0.015,B 0.000,C 180.000} C_DIS
LIN {X -227.565,Y 332.478,Z -40.000,A 0.015,B 0.000,C 180.000} C_DIS
LIN {X -228.065,Y 332.099,Z -40.000,A 0.015,B -0.000,C 180.000} C_DIS
LIN {X -229.516,Y 330.768,Z -40.000,A 0.015,B 0.000,C -180.000} C_DIS
LIN {X -229.558,Y 330.729,Z -40.000,A 0.015,B -0.000,C 180.000} C_DIS
LIN {X -236.639,Y 324.009,Z -40.000,A 0.015,B 0.000,C 180.000} C_DIS
LIN {X -236.935,Y 323.690,Z -40.000,A 0.015,B 0.000,C 180.000} C_DIS
LIN {X -237.820,Y 322.602,Z -40.000,A 0.015,B -0.000,C -180.000} C_DIS
LIN {X -238.117,Y 322.172,Z -40.000,A 0.015,B 0.000,C -180.000} C_DIS
LIN {X -240.445,Y 318.182,Z -40.000,A 0.015,B 0.000,C -180.000} C_DIS
LIN {X -240.488,Y 318.106,Z -40.000,A 0.015,B 0.000,C 180.000} C_DIS
LIN {X -243.677,Y 312.302,Z -40.000,A 0.015,B 0.000,C -180.000} C_DIS
LIN {X -243.844,Y 311.953,Z -40.000,A 0.015,B -0.000,C 180.000} C_DIS
LIN {X -244.733,Y 309.777,Z -40.000,A 0.015,B 0.000,C 180.000} C_DIS
LIN {X -244.946,Y 309.009,Z -40.000,A 0.015,B -0.000,C -180.000} C_DIS
LIN {X -246.389,Y 299.577,Z -40.000,A 0.015,B 0.000,C 180.000} C_DIS
LIN {X -246.415,Y 299.356,Z -40.000,A 0.015,B 0.000,C 180.000} C_DIS
LIN {X -246.509,Y 298.268,Z -40.000,A 0.015,B 0.000,C -180.000} C_DIS
CIRC {X -246.514,Y 297.751,Z -40.000,A 0.015,B 0.000,C -180.000},{X -246.441,Y 297.240,Z -40.000,A 0.015,B 0.000,C -180.000} C_DIS
LIN {X -245.042,Y 290.982,Z -40.000,A 0.015,B -0.000,C 180.000} C_DIS
LIN {X -245.027,Y 290.915,Z -40.000,A 0.015,B 0.000,C 180.000} C_DIS
LIN {X -244.072,Y 287.016,Z -40.000,A 0.015,B -0.000,C 180.000} C_DIS
LIN {X -243.747,Y 286.184,Z -40.000,A 0.015,B 0.000,C 180.000} C_DIS
LIN {X -241.424,Y 281.983,Z -40.000,A 0.015,B 0.000,C -180.000} C_DIS
LIN {X -241.223,Y 281.662,Z -40.000,A 0.015,B 0.000,C -180.000} C_DIS
LIN {X -240.293,Y 280.352,Z -40.000,A 0.015,B 0.000,C 180.000} C_DIS
LIN {X -240.105,Y 280.111,Z -40.000,A 0.015,B 0.000,C -180.000} C_DIS
LIN {X -237.064,Y 276.554,Z -40.000,A 0.015,B 0.000,C 180.000} C_DIS
LIN {X -236.752,Y 276.234,Z -40.000,A 0.015,B 0.000,C 180.000} C_DIS
LIN {X -236.387,Y 275.907,Z -40.000,A 0.015,B 0.000,C 180.000} C_DIS
LIN {X -236.118,Y 275.689,Z -40.000,A 0.015,B -0.000,C -180.000} C_DIS
LIN {X -230.670,Y 271.729,Z -40.000,A 0.015,B 0.000,C -180.000} C_DIS
LIN {X -230.195,Y 271.440,Z -40.000,A 0.015,B 0.000,C 180.000} C_DIS
LIN {X -227.166,Y 269.923,Z -40.000,A 0.015,B -0.000,C -180.000} C_DIS
LIN {X -226.742,Y 269.746,Z -40.000,A 0.015,B 0.000,C 180.000} C_DIS
LIN {X -223.241,Y 268.554,Z -40.000,A 0.015,B 0.000,C 180.000} C_DIS
LIN {X -222.617,Y 268.406,Z -40.000,A 0.015,B 0.000,C -180.000} C_DIS
LIN {X -215.361,Y 267.397,Z -40.000,A 0.015,B 0.000,C -180.000} C_DIS
LIN {X -214.895,Y 267.364,Z -40.000,A 0.015,B -0.000,C -180.000} C_DIS
LIN {X -178.617,Y 267.364,Z -40.000,A 0.015,B -0.000,C -180.000} C_DIS
LIN {X -178.150,Y 267.397,Z -40.000,A 0.015,B 0.000,C -180.000} C_DIS
LIN {X -170.895,Y 268.406,Z -40.000,A 0.015,B -0.000,C 180.000} C_DIS
LIN {X -170.314,Y 268.540,Z -40.000,A 0.015,B 0.000,C 180.000} C_DIS
LIN {X -167.475,Y 269.464,Z -40.000,A 0.015,B 0.000,C -180.000} C_DIS
LIN {X -167.104,Y 269.609,Z -40.000,A 0.015,B 0.000,C -180.000} C_DIS
LIN {X -164.138,Y 270.979,Z -40.000,A 0.015,B 0.000,C 180.000} C_DIS
LIN {X -163.711,Y 271.215,Z -40.000,A 0.015,B 0.000,C -180.000} C_DIS
LIN {X -161.535,Y 272.631,Z -40.000,A 0.015,B 0.000,C 180.000} C_DIS
LIN {X -161.344,Y 272.765,Z -40.000,A 0.015,B 0.000,C 180.000} C_DIS
LIN {X -156.983,Y 276.051,Z -40.000,A 0.015,B -0.000,C -180.000} C_DIS
LIN {X -156.449,Y 276.553,Z -40.000,A 0.015,B 0.000,C -180.000} C_DIS
LIN {X -153.965,Y 279.455,Z -40.000,A 0.015,B 0.000,C -180.000} C_DIS
LIN {X -153.838,Y 279.613,Z -40.000,A 0.015,B -0.000,C 180.000} C_DIS
LIN {X -152.350,Y 281.579,Z -40.000,A 0.015,B -0.000,C -180.000} C_DIS
LIN {X -152.088,Y 281.983,Z -40.000,A 0.015,B 0.000,C 180.000} C_DIS
LIN {X -149.765,Y 286.184,Z -40.000,A 0.015,B 0.000,C -180.000} C_DIS
LIN {X -149.434,Y 287.041,Z -40.000,A 0.015,B 0.000,C -180.000} C_DIS
LIN {X -147.116,Y 296.836,Z -40.000,A 0.015,B -0.000,C 180.000} C_DIS
LIN {X -147.029,Y 297.456,Z -40.000,A 0.015,B 0.000,C -180.000} C_DIS
LIN {X -146.995,Y 298.182,Z -40.000,A 0.015,B 0.000,C 180.000} C_DIS
LIN {X -147.027,Y 298.837,Z -40.000,A 0.015,B -0.000,C 180.000} C_DIS
LIN {X -148.481,Y 308.631,Z -40.000,A 0.015,B 0.000,C 180.000} C_DIS
LIN {X -148.629,Y 309.238,Z -40.000,A 0.015,B -0.000,C 180.000} C_DIS
LIN {X -149.256,Y 311.052,Z -40.000,A 0.015,B -0.000,C 180.000} C_DIS
LIN {X -149.459,Y 311.523,Z -40.000,A 0.015,B -0.000,C 180.000} C_DIS
LIN {X -151.368,Y 315.150,Z -40.000,A 0.015,B -0.000,C -180.000} C_DIS
LIN {X -151.420,Y 315.246,Z -40.000,A 0.015,B 0.000,C -180.000} C_DIS
LIN {X -155.128,Y 321.775,Z -40.000,A 0.015,B -0.000,C 180.000} C_DIS
LIN {X -155.367,Y 322.139,Z -40.000,A 0.015,B -0.000,C 180.000} C_DIS
LIN {X -156.186,Y 323.227,Z -40.000,A 0.015,B 0.000,C -180.000} C_DIS
LIN {X -156.466,Y 323.554,Z -40.000,A 0.015,B 0.000,C 180.000} C_DIS
LIN {X -157.527,Y 324.642,Z -40.000,A 0.015,B 0.000,C 180.000} C_DIS
LIN {X -157.627,Y 324.741,Z -40.000,A 0.015,B -0.000,C 180.000} C_DIS
LIN {X -165.048,Y 331.747,Z -40.000,A 0.015,B 0.000,C 180.000} C_DIS
LIN {X -165.399,Y 332.036,Z -40.000,A 0.015,B -0.000,C 180.000} C_DIS
LIN {X -166.850,Y 333.076,Z -40.000,A 0.015,B 0.000,C 180.000} C_DIS
LIN {X -167.339,Y 333.368,Z -40.000,A 0.015,B 0.000,C -180.000} C_DIS
LIN {X -177.860,Y 338.498,Z -40.000,A 0.015,B -0.000,C 180.000} C_DIS
LIN {X -178.187,Y 338.636,Z -40.000,A 0.015,B 0.000,C -180.000} C_DIS
LIN {X -178.913,Y 338.900,Z -40.000,A 0.015,B 0.000,C 180.000} C_DIS
LIN {X -179.550,Y 339.063,Z -40.000,A 0.015,B -0.000,C 180.000} C_DIS
LIN {X -180.459,Y 339.204,Z -40.000,A 0.015,B -0.000,C 180.000} C_DIS
LIN {X 4.865,Y 339.209,Z -40.000,A 0.015,B 0.000,C -180.000} C_DIS
LIN {X 5.937,Y 339.152,Z -40.000,A 0.015,B 0.000,C -180.000} C_DIS
LIN {X 6.802,Y 338.955,Z -40.000,A 0.015,B 0.000,C 180.000} C_DIS
LIN {X 7.069,Y 338.840,Z -40.000,A 0.015,B 0.000,C 180.000} C_DIS
LIN {X 7.374,Y 338.634,Z -40.000,A 0.015,B 0.000,C 180.000} C_DIS
LIN {X 9.664,Y 336.377,Z -40.000,A 0.015,B 0.000,C -180.000} C_DIS
LIN {X 9.898,Y 336.018,Z -40.000,A 0.015,B 0.000,C 180.000} C_DIS
LIN {X 10.072,Y 335.556,Z -40.000,A 0.015,B -0.000,C -180.000} C_DIS
LIN {X 10.265,Y 334.347,Z -40.000,A 0.015,B 0.000,C -180.000} C_DIS
LIN {X 10.273,Y 31.868,Z -40.000,A 0.015,B 0.000,C 180.000} C_DIS
LIN {X 9.175,Y 36.460,Z -40.000,A 0.015,B 0.000,C 180.000} C_DIS
LIN {X 9.030,Y 36.920,Z -40.000,A 0.015,B -0.000,C 180.000} C_DIS
LIN {X 8.484,Y 38.296,Z -40.000,A 0.015,B 0.000,C 180.000} C_DIS
LIN {X 8.269,Y 38.741,Z -40.000,A 0.015,B -0.000,C 180.000} C_DIS
LIN {X 6.110,Y 42.480,Z -40.000,A 0.015,B 0.000,C 180.000} C_DIS
LIN {X 6.074,Y 42.541,Z -40.000,A 0.015,B 0.000,C -180.000} C_DIS
LIN {X 2.559,Y 48.345,Z -40.000,A 0.015,B 0.000,C -180.000} C_DIS
LIN {X 2.347,Y 48.655,Z -40.000,A 0.015,B 0.000,C 180.000} C_DIS
LIN {X 1.045,Y 50.348,Z -40.000,A 0.015,B 0.000,C 180.000} C_DIS
LIN {X 0.484,Y 50.921,Z -40.000,A 0.015,B 0.000,C 180.000} C_DIS
LIN {X -7.437,Y 57.295,Z -40.000,A 0.015,B -0.000,C -180.000} C_DIS
LIN {X -7.809,Y 57.555,Z -40.000,A 0.015,B 0.000,C 180.000} C_DIS
LIN {X -8.474,Y 57.956,Z -40.000,A 0.015,B 0.000,C 180.000} C_DIS
LIN {X -9.244,Y 58.299,Z -40.000,A 0.015,B 0.000,C -180.000} C_DIS
LIN {X -19.100,Y 61.275,Z -40.000,A 0.015,B 0.000,C 180.000} C_DIS
LIN {X -20.008,Y 61.419,Z -40.000,A 0.015,B 0.000,C -180.000} C_DIS
LIN {X -23.998,Y 61.502,Z -40.000,A 0.015,B 0.000,C 180.000} C_DIS
LIN {X -24.254,Y 61.498,Z -40.000,A 0.015,B 0.000,C -180.000} C_DIS
LIN {X -26.431,Y 61.378,Z -40.000,A 0.015,B 0.000,C 180.000} C_DIS
LIN {X -26.852,Y 61.329,Z -40.000,A 0.015,B -0.000,C 180.000} C_DIS
LIN {X -31.568,Y 60.469,Z -40.000,A 0.015,B 0.000,C -180.000} C_DIS
LIN {X -32.207,Y 60.286,Z -40.000,A 0.015,B 0.000,C -180.000} C_DIS
LIN {X -34.021,Y 59.568,Z -40.000,A 0.015,B 0.000,C 180.000} C_DIS
LIN {X -34.163,Y 59.508,Z -40.000,A 0.015,B 0.000,C -180.000} C_DIS
LIN {X -39.242,Y 57.223,Z -40.000,A 0.015,B -0.000,C -180.000} C_DIS
LIN {X -39.736,Y 56.949,Z -40.000,A 0.015,B 0.000,C 180.000} C_DIS
LIN {X -42.338,Y 55.208,Z -40.000,A 0.015,B 0.000,C 180.000} C_DIS
LIN {X -42.659,Y 54.964,Z -40.000,A 0.015,B 0.000,C 180.000} C_DIS
LIN {X -44.778,Y 53.147,Z -40.000,A 0.015,B 0.000,C 180.000} C_DIS
LIN {X -44.958,Y 52.980,Z -40.000,A 0.015,B 0.000,C -180.000} C_DIS
LIN {X -46.051,Y 51.896,Z -40.000,A 0.015,B 0.000,C 180.000} C_DIS
LIN {X -46.345,Y 51.563,Z -40.000,A 0.015,B 0.000,C 180.000} C_DIS
LIN {X -50.392,Y 46.326,Z -40.000,A 0.015,B 0.000,C 180.000} C_DIS
LIN {X -50.645,Y 45.950,Z -40.000,A 0.015,B 0.000,C 180.000} C_DIS
LIN {X -68.791,Y 14.550,Z -40.000,A 0.015,B -0.000,C 180.000} C_DIS
LIN {X -68.976,Y 14.178,Z -40.000,A 0.015,B 0.000,C -180.000} C_DIS
LIN {X -70.669,Y 10.188,Z -40.000,A 0.015,B 0.000,C -180.000} C_DIS
LIN {X -70.710,Y 10.087,Z -40.000,A 0.015,B 0.000,C -180.000} C_DIS
LIN {X -71.831,Y 7.185,Z -40.000,A 0.015,B -0.000,C 180.000} C_DIS
LIN {X -71.985,Y 6.669,Z -40.000,A 0.015,B 0.000,C 180.000} C_DIS
LIN {X -72.602,Y 3.767,Z -40.000,A 0.015,B 0.000,C -180.000} C_DIS
LIN {X -72.661,Y 3.382,Z -40.000,A 0.015,B 0.000,C 180.000} C_DIS
LIN {X -72.936,Y 0.481,Z -40.000,A 0.015,B -0.000,C 180.000} C_DIS
LIN {X -72.951,Y 0.215,Z -40.000,A 0.015,B -0.000,C -180.000} C_DIS
LIN {X -72.974,Y -1.235,Z -40.000,A 0.015,B -0.000,C -180.000} C_DIS
LIN {X -72.953,Y -1.669,Z -40.000,A 0.015,B -0.000,C 180.000} C_DIS
LIN {X -72.174,Y -8.562,Z -40.000,A 0.015,B 0.000,C 180.000} C_DIS
LIN {X -72.004,Y -9.303,Z -40.000,A 0.015,B 0.000,C -180.000} C_DIS
LIN {X -70.794,Y -12.746,Z -40.000,A 0.015,B 0.000,C 180.000} C_DIS
LIN {X -70.740,Y -12.891,Z -40.000,A 0.015,B 0.000,C -180.000} C_DIS
LIN {X -69.915,Y -14.933,Z -40.000,A 0.015,B 0.000,C -180.000} C_DIS
LIN {X -69.713,Y -15.349,Z -40.000,A 0.015,B 0.000,C -180.000} C_DIS
LIN {X -67.660,Y -18.932,Z -40.000,A 0.015,B 0.000,C 180.000} C_DIS
LIN {X -67.532,Y -19.138,Z -40.000,A 0.015,B 0.000,C 180.000} C_DIS
LIN {X -66.782,Y -20.252,Z -40.000,A 0.015,B 0.000,C 180.000} C_DIS
LIN {X -66.294,Y -20.827,Z -40.000,A 0.015,B 0.000,C -180.000} C_DIS
LIN {X -59.764,Y -26.976,Z -40.000,A 0.015,B -0.000,C 180.000} C_DIS
LIN {X -59.603,Y -27.117,Z -40.000,A 0.015,B 0.000,C -180.000} C_DIS
LIN {X -58.515,Y -28.019,Z -40.000,A 0.015,B 0.000,C 180.000} C_DIS
CIRC {X -58.083,Y -28.324,Z -40.000,A 0.015,B -0.000,C -180.000},{X -57.609,Y -28.557,Z -40.000,A 0.015,B 0.000,C -180.000} C_DIS
LIN {X -50.808,Y -31.266,Z -40.000,A 0.015,B 0.000,C 180.000} C_DIS
LIN {X -342.732,Y -31.266,Z -40.000,A 0.015,B 0.000,C -180.000} C_DIS
LIN {X -336.289,Y -28.753,Z -40.000,A 0.015,B 0.000,C 180.000} C_DIS
LIN {X -335.787,Y -28.508,Z -40.000,A 0.015,B 0.000,C 180.000} C_DIS
LIN {X -335.061,Y -28.076,Z -40.000,A 0.015,B 0.000,C 180.000} C_DIS
LIN {X -334.483,Y -27.641,Z -40.000,A 0.015,B 0.000,C -180.000} C_DIS
LIN {X -327.583,Y -21.193,Z -40.000,A 0.015,B 0.000,C -180.000} C_DIS
LIN {X -327.362,Y -20.966,Z -40.000,A 0.015,B 0.000,C 180.000} C_DIS
